SPLINE
SPL {X  -117.449, Y  +780.140, Z    +0.000, E1  +415.491, E3 -83319.411}
SPL {X  -137.837, Y  +752.727, Z    +0.000, E1  +411.385, E3 -83338.899}
SPL {X  -150.415, Y  +726.018, Z    +0.000, E1  +402.769, E3 -83347.774}
SPL {X  -156.153, Y  +706.328, Z    +0.000, E1  +392.414, E3 -83351.466}
SPL {X  -159.178, Y  +687.603, Z    +0.000, E1  +378.267, E3 -83353.444}
SPL {X  -159.915, Y  +676.399, Z    +0.000, E1  +367.484, E3 -83354.014}
SPL {X  -159.990, Y  +669.381, Z    +0.000, E1  +359.965, E3 -83354.114}
SPL {X  -159.990, Y  +666.412, Z    +0.000, E1  +352.765, E3 -83354.146}
SPL {X  -159.990, Y  +662.995, Z    +0.000, E1  +343.976, E3 -83354.248}
SPL {X  -159.990, Y  +658.179, Z    +0.000, E1  +331.312, E3 -83354.485}
SPL {X  -159.990, Y  +652.822, Z    +0.000, E1  +319.345, E3 -83354.899}
SPL {X  -159.990, Y  +646.185, Z    +0.000, E1  +308.728, E3 -83355.638}
SPL {X  -159.990, Y  +632.371, Z    +0.000, E1  +297.040, E3 -83357.991}
SPL {X  -159.990, Y  +579.000, Z    +0.000, E1  +286.931, E3 -83372.863}
SPL {X  -157.725, Y  +355.675, Z    +0.000, E1  +284.959, E3 -83469.821}
SPL {X  -142.593, Y  +309.947, Z    +0.000, E1  +282.426, E3 -83463.485}
SPL {X  -142.198, Y  +309.176, Z    +0.000, E1  +283.218, E3 -83472.293}
ENDSPLINE

SPLINE
SPL {X  -142.352, Y  +309.474, Z    +0.000, E1  +284.206, E3 -83481.987}
ENDSPLINE

SPLINE
SPL {X  -141.553, Y  +307.937, Z    +0.000, E1  +285.290, E3 -83493.003}
SPL {X  -140.562, Y  +306.086, Z    +0.000, E1  +286.440, E3 -83503.697}
SPL {X  -138.743, Y  +302.832, Z    +0.000, E1  +287.062, E3 -83510.494}
SPL {X  -135.531, Y  +297.482, Z    +0.000, E1  +287.444, E3 -83516.329}
SPL {X  -132.271, Y  +292.493, Z    +0.000, E1  +287.844, E3 -83521.847}
SPL {X  -128.837, Y  +287.643, Z    +0.000, E1  +288.283, E3 -83527.285}
SPL {X  -125.941, Y  +283.830, Z    +0.000, E1  +288.683, E3 -83531.584}
SPL {X  -122.669, Y  +279.791, Z    +0.000, E1  +289.119, E3 -83536.078}
SPL {X  -119.730, Y  +276.380, Z    +0.000, E1  +289.584, E3 -83539.866}
SPL {X   -74.058, Y  +240.683, Z    +0.000, E1  +305.011, E3 -83695.582}
ENDSPLINE

SPLINE
SPL {X  -130.401, Y  +289.805, Z    +0.000, E1  +307.505, E3 -83852.553}
SPL {X  -152.244, Y  +333.323, Z    +0.000, E1  +320.871, E3 -83869.365}
SPL {X  -158.218, Y  +358.753, Z    +0.000, E1  +336.397, E3 -83873.537}
SPL {X  -159.681, Y  +372.564, Z    +0.000, E1  +347.981, E3 -83874.589}
SPL {X  -159.987, Y  +381.561, Z    +0.000, E1  +356.806, E3 -83874.885}
SPL {X  -159.990, Y  +384.668, Z    +0.000, E1  +360.183, E3 -83874.911}
SPL {X  -159.990, Y  +387.837, Z    +0.000, E1  +367.342, E3 -83874.951}
SPL {X  -159.990, Y  +393.084, Z    +0.000, E1  +380.137, E3 -83875.161}
SPL {X  -159.990, Y  +401.914, Z    +0.000, E1  +400.147, E3 -83875.855}
SPL {X  -159.990, Y  +414.609, Z    +0.000, E1  +416.791, E3 -83877.592}
SPL {X  -159.990, Y  +464.476, Z    +0.000, E1  +431.765, E3 -83890.393}
SPL {X  -157.643, Y  +698.802, Z    +0.000, E1  +434.751, E3 -83993.407}
SPL {X  -154.470, Y  +713.164, Z    +0.000, E1  +434.425, E3 -84004.996}
SPL {X  -151.032, Y  +724.285, Z    +0.000, E1  +434.102, E3 -84014.800}
SPL {X  -147.134, Y  +734.337, Z    +0.000, E1  +433.686, E3 -84024.437}
SPL {X  -143.804, Y  +741.622, Z    +0.000, E1  +433.324, E3 -84031.825}
SPL {X  -140.603, Y  +747.839, Z    +0.000, E1  +432.964, E3 -84038.341}
SPL {X  -137.184, Y  +753.824, Z    +0.000, E1  +432.574, E3 -84044.778}
SPL {X  -133.762, Y  +759.276, Z    +0.000, E1  +432.150, E3 -84050.831}
SPL {X  -130.927, Y  +763.451, Z    +0.000, E1  +431.785, E3 -84055.526}
SPL {X  -126.852, Y  +768.996, Z    +0.000, E1  +431.276, E3 -84061.757}
SPL {X  -122.512, Y  +774.396, Z    +0.000, E1  +430.640, E3 -84067.866}
SPL {X  -119.782, Y  +777.562, Z    +0.000, E1  +430.221, E3 -84071.373}
SPL {X   -71.924, Y  +814.412, Z    +0.000, E1  +415.124, E3 -84228.243}
ENDSPLINE

SPLINE
SPL {X  -132.255, Y  +761.530, Z    +0.000, E1  +413.203, E3 -84391.413}
SPL {X  -150.415, Y  +726.018, Z    +0.000, E1  +402.769, E3 -84404.917}
SPL {X  -156.153, Y  +706.328, Z    +0.000, E1  +392.414, E3 -84408.609}
SPL {X  -159.178, Y  +687.603, Z    +0.000, E1  +378.267, E3 -84410.587}
SPL {X  -159.974, Y  +673.783, Z    +0.000, E1  +364.843, E3 -84411.209}
SPL {X  -159.990, Y  +669.500, Z    +0.000, E1  +360.000, E3 -84411.256}
SPL {X  -159.990, Y  +667.470, Z    +0.000, E1  +355.588, E3 -84411.274}
SPL {X  -159.990, Y  +662.995, Z    +0.000, E1  +343.976, E3 -84411.391}
SPL {X  -159.990, Y  +658.179, Z    +0.000, E1  +331.312, E3 -84411.628}
SPL {X  -159.990, Y  +652.822, Z    +0.000, E1  +319.345, E3 -84412.042}
SPL {X  -159.990, Y  +646.185, Z    +0.000, E1  +308.728, E3 -84412.781}
SPL {X  -159.990, Y  +632.371, Z    +0.000, E1  +297.040, E3 -84415.134}
SPL {X  -159.990, Y  +579.000, Z    +0.000, E1  +286.931, E3 -84430.006}
SPL {X  -157.725, Y  +355.675, Z    +0.000, E1  +284.959, E3 -84526.964}
SPL {X  -142.593, Y  +309.947, Z    +0.000, E1  +282.426, E3 -84520.628}
SPL {X  -142.198, Y  +309.176, Z    +0.000, E1  +283.218, E3 -84529.436}
ENDSPLINE

SPLINE
SPL {X  -142.352, Y  +309.474, Z    +0.000, E1  +284.206, E3 -84539.130}
ENDSPLINE

SPLINE
SPL {X  -141.553, Y  +307.937, Z    +0.000, E1  +285.290, E3 -84550.146}
SPL {X  -140.562, Y  +306.086, Z    +0.000, E1  +286.440, E3 -84560.839}
SPL {X  -138.743, Y  +302.832, Z    +0.000, E1  +287.062, E3 -84567.637}
SPL {X  -135.531, Y  +297.482, Z    +0.000, E1  +287.444, E3 -84573.471}
SPL {X  -132.271, Y  +292.493, Z    +0.000, E1  +287.844, E3 -84578.990}
SPL {X  -128.837, Y  +287.643, Z    +0.000, E1  +288.283, E3 -84584.428}
SPL {X  -124.965, Y  +282.598, Z    +0.000, E1  +288.800, E3 -84590.089}
SPL {X  -120.791, Y  +277.589, Z    +0.000, E1  +289.397, E3 -84595.662}
SPL {X   -74.058, Y  +240.683, Z    +0.000, E1  +305.011, E3 -84752.725}
ENDSPLINE

SPLINE
SPL {X  -130.401, Y  +289.805, Z    +0.000, E1  +307.505, E3 -84909.696}
SPL {X  -148.502, Y  +322.968, Z    +0.000, E1  +316.497, E3 -84924.016}
SPL {X  -154.800, Y  +342.080, Z    +0.000, E1  +325.471, E3 -84928.320}
SPL {X  -158.218, Y  +358.753, Z    +0.000, E1  +336.397, E3 -84930.680}
SPL {X  -159.681, Y  +372.564, Z    +0.000, E1  +347.981, E3 -84931.731}
SPL {X  -159.987, Y  +381.561, Z    +0.000, E1  +356.806, E3 -84932.028}
SPL {X  -159.990, Y  +384.668, Z    +0.000, E1  +360.183, E3 -84932.054}
SPL {X  -159.990, Y  +387.837, Z    +0.000, E1  +367.342, E3 -84932.094}
SPL {X  -159.990, Y  +393.084, Z    +0.000, E1  +380.137, E3 -84932.304}
SPL {X  -159.990, Y  +401.914, Z    +0.000, E1  +400.147, E3 -84932.998}
SPL {X  -159.990, Y  +414.609, Z    +0.000, E1  +416.791, E3 -84934.735}
SPL {X  -159.990, Y  +464.476, Z    +0.000, E1  +431.765, E3 -84947.536}
SPL {X  -157.643, Y  +698.802, Z    +0.000, E1  +434.751, E3 -85050.550}
SPL {X  -154.470, Y  +713.164, Z    +0.000, E1  +434.425, E3 -85062.139}
SPL {X  -151.032, Y  +724.285, Z    +0.000, E1  +434.102, E3 -85071.943}
SPL {X  -147.134, Y  +734.337, Z    +0.000, E1  +433.686, E3 -85081.580}
SPL {X  -143.804, Y  +741.622, Z    +0.000, E1  +433.324, E3 -85088.968}
SPL {X  -140.603, Y  +747.839, Z    +0.000, E1  +432.964, E3 -85095.484}
SPL {X  -137.184, Y  +753.824, Z    +0.000, E1  +432.574, E3 -85101.920}
SPL {X  -133.762, Y  +759.276, Z    +0.000, E1  +432.150, E3 -85107.974}
SPL {X  -130.927, Y  +763.451, Z    +0.000, E1  +431.785, E3 -85112.669}
SPL {X  -126.852, Y  +768.996, Z    +0.000, E1  +431.276, E3 -85118.900}
SPL {X  -122.512, Y  +774.396, Z    +0.000, E1  +430.640, E3 -85125.009}
SPL {X  -119.782, Y  +777.562, Z    +0.000, E1  +430.221, E3 -85128.516}
SPL {X   -71.924, Y  +814.412, Z    +0.000, E1  +415.124, E3 -85285.386}
ENDSPLINE

SPLINE
SPL {X  -132.255, Y  +761.530, Z    +0.000, E1  +413.203, E3 -85448.556}
SPL {X  -150.415, Y  +726.018, Z    +0.000, E1  +402.769, E3 -85462.060}
SPL {X  -156.153, Y  +706.328, Z    +0.000, E1  +392.414, E3 -85465.752}
SPL {X  -159.178, Y  +687.603, Z    +0.000, E1  +378.267, E3 -85467.730}
SPL {X  -159.915, Y  +676.399, Z    +0.000, E1  +367.484, E3 -85468.300}
SPL {X  -159.990, Y  +669.585, Z    +0.000, E1  +360.185, E3 -85468.399}
SPL {X  -159.990, Y  +667.470, Z    +0.000, E1  +355.588, E3 -85468.417}
SPL {X  -159.990, Y  +662.995, Z    +0.000, E1  +343.976, E3 -85468.534}
SPL {X  -159.990, Y  +658.179, Z    +0.000, E1  +331.312, E3 -85468.770}
SPL {X  -159.990, Y  +652.822, Z    +0.000, E1  +319.345, E3 -85469.185}
SPL {X  -159.990, Y  +646.185, Z    +0.000, E1  +308.728, E3 -85469.924}
SPL {X  -159.990, Y  +632.371, Z    +0.000, E1  +297.040, E3 -85472.276}
SPL {X  -159.990, Y  +579.000, Z    +0.000, E1  +286.931, E3 -85487.149}
SPL {X  -157.725, Y  +355.675, Z    +0.000, E1  +284.959, E3 -85584.107}
SPL {X  -142.593, Y  +309.947, Z    +0.000, E1  +282.426, E3 -85577.770}
SPL {X  -142.198, Y  +309.176, Z    +0.000, E1  +283.218, E3 -85586.579}
ENDSPLINE

SPLINE
SPL {X  -142.352, Y  +309.474, Z    +0.000, E1  +284.206, E3 -85596.273}
ENDSPLINE

SPLINE
SPL {X  -141.553, Y  +307.937, Z    +0.000, E1  +285.290, E3 -85607.288}
SPL {X  -140.562, Y  +306.086, Z    +0.000, E1  +286.440, E3 -85617.982}
SPL {X  -138.743, Y  +302.832, Z    +0.000, E1  +287.062, E3 -85624.780}
SPL {X  -135.531, Y  +297.482, Z    +0.000, E1  +287.444, E3 -85630.614}
SPL {X  -132.271, Y  +292.493, Z    +0.000, E1  +287.844, E3 -85636.133}
SPL {X  -128.837, Y  +287.643, Z    +0.000, E1  +288.283, E3 -85641.570}
SPL {X  -124.965, Y  +282.598, Z    +0.000, E1  +288.800, E3 -85647.232}
SPL {X  -120.791, Y  +277.589, Z    +0.000, E1  +289.397, E3 -85652.805}
SPL {X   -74.058, Y  +240.683, Z    +0.000, E1  +305.011, E3 -85809.868}
ENDSPLINE

SPLINE
SPL {X  -130.401, Y  +289.805, Z    +0.000, E1  +307.505, E3 -85966.839}
SPL {X  -148.502, Y  +322.968, Z    +0.000, E1  +316.497, E3 -85981.159}
SPL {X  -154.800, Y  +342.080, Z    +0.000, E1  +325.471, E3 -85985.463}
SPL {X  -158.218, Y  +358.753, Z    +0.000, E1  +336.397, E3 -85987.823}
SPL {X  -159.681, Y  +372.564, Z    +0.000, E1  +347.981, E3 -85988.874}
SPL {X  -159.987, Y  +381.561, Z    +0.000, E1  +356.806, E3 -85989.171}
SPL {X  -159.990, Y  +384.668, Z    +0.000, E1  +360.183, E3 -85989.196}
SPL {X  -159.990, Y  +387.837, Z    +0.000, E1  +367.342, E3 -85989.237}
SPL {X  -159.990, Y  +393.084, Z    +0.000, E1  +380.137, E3 -85989.447}
SPL {X  -159.990, Y  +401.914, Z    +0.000, E1  +400.147, E3 -85990.141}
SPL {X  -159.990, Y  +414.609, Z    +0.000, E1  +416.791, E3 -85991.877}
SPL {X  -159.990, Y  +464.476, Z    +0.000, E1  +431.765, E3 -86004.678}
SPL {X  -157.643, Y  +698.802, Z    +0.000, E1  +434.751, E3 -86107.693}
SPL {X  -154.470, Y  +713.164, Z    +0.000, E1  +434.425, E3 -86119.282}
SPL {X  -151.032, Y  +724.285, Z    +0.000, E1  +434.102, E3 -86129.086}
SPL {X  -147.134, Y  +734.337, Z    +0.000, E1  +433.686, E3 -86138.723}
SPL {X  -143.804, Y  +741.622, Z    +0.000, E1  +433.324, E3 -86146.111}
SPL {X  -140.603, Y  +747.839, Z    +0.000, E1  +432.964, E3 -86152.627}
SPL {X  -137.184, Y  +753.824, Z    +0.000, E1  +432.574, E3 -86159.063}
SPL {X  -133.762, Y  +759.276, Z    +0.000, E1  +432.150, E3 -86165.117}
SPL {X  -130.927, Y  +763.451, Z    +0.000, E1  +431.785, E3 -86169.812}
SPL {X  -128.105, Y  +767.343, Z    +0.000, E1  +431.419, E3 -86174.200}
SPL {X  -124.554, Y  +771.914, Z    +0.000, E1  +430.935, E3 -86179.371}
SPL {X  -120.687, Y  +776.531, Z    +0.000, E1  +430.379, E3 -86184.505}
SPL {X   -71.924, Y  +814.412, Z    +0.000, E1  +415.124, E3 -86342.529}
ENDSPLINE

SPLINE
SPL {X  -132.255, Y  +761.530, Z    +0.000, E1  +413.203, E3 -86505.699}
SPL {X  -150.415, Y  +726.018, Z    +0.000, E1  +402.769, E3 -86519.203}
SPL {X  -156.153, Y  +706.328, Z    +0.000, E1  +392.414, E3 -86522.895}
SPL {X  -159.178, Y  +687.603, Z    +0.000, E1  +378.267, E3 -86524.873}
SPL {X  -159.974, Y  +673.783, Z    +0.000, E1  +364.843, E3 -86525.495}
SPL {X  -159.990, Y  +669.500, Z    +0.000, E1  +360.000, E3 -86525.542}
SPL {X  -159.990, Y  +667.470, Z    +0.000, E1  +355.588, E3 -86525.560}
SPL {X  -159.990, Y  +662.995, Z    +0.000, E1  +343.976, E3 -86525.677}
SPL {X  -159.990, Y  +658.179, Z    +0.000, E1  +331.312, E3 -86525.913}
SPL {X  -159.990, Y  +652.822, Z    +0.000, E1  +319.345, E3 -86526.328}
SPL {X  -159.990, Y  +646.185, Z    +0.000, E1  +308.728, E3 -86527.067}
SPL {X  -159.990, Y  +636.375, Z    +0.000, E1  +299.286, E3 -86528.506}
SPL {X  -159.990, Y  +617.374, Z    +0.000, E1  +291.478, E3 -86532.833}
SPL {X  -159.990, Y  +579.000, Z    +0.000, E1  +286.931, E3 -86544.292}
SPL {X  -157.725, Y  +355.675, Z    +0.000, E1  +284.959, E3 -86641.250}
SPL {X  -142.593, Y  +309.947, Z    +0.000, E1  +282.426, E3 -86634.913}
SPL {X  -142.198, Y  +309.176, Z    +0.000, E1  +283.218, E3 -86643.722}
ENDSPLINE

SPLINE
SPL {X  -142.352, Y  +309.474, Z    +0.000, E1  +284.206, E3 -86653.415}
ENDSPLINE

SPLINE
SPL {X  -141.929, Y  +308.657, Z    +0.000, E1  +285.131, E3 -86662.501}
SPL {X  -140.635, Y  +306.221, Z    +0.000, E1  +286.163, E3 -86672.913}
SPL {X  -138.743, Y  +302.832, Z    +0.000, E1  +287.062, E3 -86681.923}
SPL {X  -135.531, Y  +297.482, Z    +0.000, E1  +287.444, E3 -86687.757}
SPL {X  -132.271, Y  +292.493, Z    +0.000, E1  +287.844, E3 -86693.276}
SPL {X  -128.837, Y  +287.643, Z    +0.000, E1  +288.283, E3 -86698.713}
SPL {X  -125.941, Y  +283.830, Z    +0.000, E1  +288.683, E3 -86703.013}
SPL {X  -124.080, Y  +281.501, Z    +0.000, E1  +288.943, E3 -86705.624}
SPL {X  -120.791, Y  +277.589, Z    +0.000, E1  +289.397, E3 -86709.948}
SPL {X   -74.058, Y  +240.683, Z    +0.000, E1  +305.011, E3 -86867.011}
ENDSPLINE

SPLINE
SPL {X  -130.401, Y  +289.805, Z    +0.000, E1  +307.505, E3 -87023.982}
SPL {X  -152.244, Y  +333.323, Z    +0.000, E1  +320.871, E3 -87040.793}
SPL {X  -158.218, Y  +358.753, Z    +0.000, E1  +336.397, E3 -87044.966}
SPL {X  -159.681, Y  +372.564, Z    +0.000, E1  +347.981, E3 -87046.017}
SPL {X  -159.987, Y  +381.561, Z    +0.000, E1  +356.806, E3 -87046.314}
SPL {X  -159.990, Y  +384.668, Z    +0.000, E1  +360.183, E3 -87046.339}
SPL {X  -159.990, Y  +387.837, Z    +0.000, E1  +367.342, E3 -87046.380}
SPL {X  -159.990, Y  +393.084, Z    +0.000, E1  +380.137, E3 -87046.590}
SPL {X  -159.990, Y  +401.914, Z    +0.000, E1  +400.147, E3 -87047.283}
SPL {X  -159.990, Y  +414.609, Z    +0.000, E1  +416.791, E3 -87049.020}
SPL {X  -159.990, Y  +464.476, Z    +0.000, E1  +431.765, E3 -87061.821}
SPL {X  -158.553, Y  +692.895, Z    +0.000, E1  +434.809, E3 -87160.585}
SPL {X  -156.740, Y  +703.585, Z    +0.000, E1  +434.640, E3 -87168.589}
SPL {X  -154.470, Y  +713.164, Z    +0.000, E1  +434.425, E3 -87176.425}
SPL {X  -151.032, Y  +724.285, Z    +0.000, E1  +434.102, E3 -87186.228}
SPL {X  -147.134, Y  +734.337, Z    +0.000, E1  +433.686, E3 -87195.866}
SPL {X  -143.804, Y  +741.622, Z    +0.000, E1  +433.324, E3 -87203.254}
SPL {X  -140.603, Y  +747.839, Z    +0.000, E1  +432.964, E3 -87209.769}
SPL {X  -137.184, Y  +753.824, Z    +0.000, E1  +432.574, E3 -87216.206}
SPL {X  -133.762, Y  +759.276, Z    +0.000, E1  +432.150, E3 -87222.260}
SPL {X  -130.927, Y  +763.451, Z    +0.000, E1  +431.785, E3 -87226.954}
SPL {X  -126.852, Y  +768.996, Z    +0.000, E1  +431.276, E3 -87233.185}
SPL {X  -122.512, Y  +774.396, Z    +0.000, E1  +430.640, E3 -87239.295}
SPL {X  -119.782, Y  +777.562, Z    +0.000, E1  +430.221, E3 -87242.802}
SPL {X   -71.924, Y  +814.412, Z    +0.000, E1  +415.124, E3 -87399.672}
ENDSPLINE

SPLINE
SPL {X  -132.255, Y  +761.530, Z    +0.000, E1  +413.203, E3 -87562.842}
SPL {X  -150.415, Y  +726.018, Z    +0.000, E1  +402.769, E3 -87576.346}
SPL {X  -156.153, Y  +706.328, Z    +0.000, E1  +392.414, E3 -87580.038}
SPL {X  -159.178, Y  +687.603, Z    +0.000, E1  +378.267, E3 -87582.016}
SPL {X  -159.974, Y  +673.783, Z    +0.000, E1  +364.843, E3 -87582.637}
SPL {X  -159.990, Y  +669.500, Z    +0.000, E1  +360.000, E3 -87582.685}
SPL {X  -159.990, Y  +667.470, Z    +0.000, E1  +355.588, E3 -87582.703}
SPL {X  -159.990, Y  +662.995, Z    +0.000, E1  +343.976, E3 -87582.819}
SPL {X  -159.990, Y  +658.179, Z    +0.000, E1  +331.312, E3 -87583.056}
SPL {X  -159.990, Y  +652.822, Z    +0.000, E1  +319.345, E3 -87583.471}
SPL {X  -159.990, Y  +646.185, Z    +0.000, E1  +308.728, E3 -87584.210}
SPL {X  -159.990, Y  +636.375, Z    +0.000, E1  +299.286, E3 -87585.649}
SPL {X  -159.990, Y  +617.374, Z    +0.000, E1  +291.478, E3 -87589.975}
SPL {X  -159.990, Y  +579.000, Z    +0.000, E1  +286.931, E3 -87601.434}
SPL {X  -157.725, Y  +355.675, Z    +0.000, E1  +284.959, E3 -87698.393}
SPL {X  -142.593, Y  +309.947, Z    +0.000, E1  +282.426, E3 -87692.056}
SPL {X  -142.198, Y  +309.176, Z    +0.000, E1  +283.218, E3 -87700.865}
ENDSPLINE

SPLINE
SPL {X  -142.352, Y  +309.474, Z    +0.000, E1  +284.206, E3 -87710.558}
ENDSPLINE

SPLINE
SPL {X  -141.553, Y  +307.937, Z    +0.000, E1  +285.290, E3 -87721.574}
SPL {X  -140.562, Y  +306.086, Z    +0.000, E1  +286.440, E3 -87732.268}
SPL {X  -138.743, Y  +302.832, Z    +0.000, E1  +287.062, E3 -87739.065}
SPL {X  -135.531, Y  +297.482, Z    +0.000, E1  +287.444, E3 -87744.900}
SPL {X  -132.271, Y  +292.493, Z    +0.000, E1  +287.844, E3 -87750.418}
SPL {X  -128.837, Y  +287.643, Z    +0.000, E1  +288.283, E3 -87755.856}
SPL {X  -125.941, Y  +283.830, Z    +0.000, E1  +288.683, E3 -87760.156}
SPL {X  -124.080, Y  +281.501, Z    +0.000, E1  +288.943, E3 -87762.766}
SPL {X  -120.791, Y  +277.589, Z    +0.000, E1  +289.397, E3 -87767.091}
SPL {X   -74.058, Y  +240.683, Z    +0.000, E1  +305.011, E3 -87924.154}
ENDSPLINE

SPLINE
SPL {X  -130.401, Y  +289.805, Z    +0.000, E1  +307.505, E3 -88081.125}
SPL {X  -148.502, Y  +322.968, Z    +0.000, E1  +316.497, E3 -88095.445}
SPL {X  -154.800, Y  +342.080, Z    +0.000, E1  +325.471, E3 -88099.749}
SPL {X  -158.218, Y  +358.753, Z    +0.000, E1  +336.397, E3 -88102.108}
SPL {X  -159.681, Y  +372.564, Z    +0.000, E1  +347.981, E3 -88103.160}
SPL {X  -159.987, Y  +381.561, Z    +0.000, E1  +356.806, E3 -88103.456}
SPL {X  -159.990, Y  +384.668, Z    +0.000, E1  +360.183, E3 -88103.482}
SPL {X  -159.990, Y  +387.837, Z    +0.000, E1  +367.342, E3 -88103.523}
SPL {X  -159.990, Y  +393.084, Z    +0.000, E1  +380.137, E3 -88103.733}
SPL {X  -159.990, Y  +401.914, Z    +0.000, E1  +400.147, E3 -88104.426}
SPL {X  -159.990, Y  +414.609, Z    +0.000, E1  +416.791, E3 -88106.163}
SPL {X  -159.990, Y  +464.476, Z    +0.000, E1  +431.765, E3 -88118.964}
SPL {X  -157.643, Y  +698.802, Z    +0.000, E1  +434.751, E3 -88221.979}
SPL {X  -154.470, Y  +713.164, Z    +0.000, E1  +434.425, E3 -88233.568}
SPL {X  -152.098, Y  +721.129, Z    +0.000, E1  +434.190, E3 -88240.540}
SPL {X  -148.128, Y  +731.956, Z    +0.000, E1  +433.814, E3 -88250.621}
SPL {X  -143.804, Y  +741.622, Z    +0.000, E1  +433.324, E3 -88260.397}
SPL {X  -140.603, Y  +747.839, Z    +0.000, E1  +432.964, E3 -88266.912}
SPL {X  -137.184, Y  +753.824, Z    +0.000, E1  +432.574, E3 -88273.349}
SPL {X  -133.762, Y  +759.276, Z    +0.000, E1  +432.150, E3 -88279.403}
SPL {X  -130.927, Y  +763.451, Z    +0.000, E1  +431.785, E3 -88284.097}
SPL {X  -128.105, Y  +767.343, Z    +0.000, E1  +431.419, E3 -88288.486}
SPL {X  -124.554, Y  +771.914, Z    +0.000, E1  +430.935, E3 -88293.657}
SPL {X  -120.687, Y  +776.531, Z    +0.000, E1  +430.379, E3 -88298.790}
SPL {X   -71.924, Y  +814.412, Z    +0.000, E1  +415.124, E3 -88456.815}
ENDSPLINE

SPLINE
SPL {X  -132.255, Y  +761.530, Z    +0.000, E1  +413.203, E3 -88619.984}
SPL {X  -150.415, Y  +726.018, Z    +0.000, E1  +402.769, E3 -88633.488}
SPL {X  -157.206, Y  +701.216, Z    +0.000, E1  +389.056, E3 -88637.827}
SPL {X  -159.772, Y  +679.843, Z    +0.000, E1  +371.089, E3 -88639.591}
SPL {X  -159.990, Y  +669.381, Z    +0.000, E1  +359.965, E3 -88639.828}
SPL {X  -159.990, Y  +666.412, Z    +0.000, E1  +352.765, E3 -88639.860}
SPL {X  -159.990, Y  +662.995, Z    +0.000, E1  +343.976, E3 -88639.962}
SPL {X  -159.990, Y  +658.179, Z    +0.000, E1  +331.312, E3 -88640.199}
SPL {X  -159.990, Y  +652.822, Z    +0.000, E1  +319.345, E3 -88640.614}
SPL {X  -159.990, Y  +646.185, Z    +0.000, E1  +308.728, E3 -88641.352}
SPL {X  -159.990, Y  +632.371, Z    +0.000, E1  +297.040, E3 -88643.705}
SPL {X  -159.990, Y  +579.000, Z    +0.000, E1  +286.931, E3 -88658.577}
SPL {X  -157.725, Y  +355.675, Z    +0.000, E1  +284.959, E3 -88755.536}
SPL {X  -142.593, Y  +309.947, Z    +0.000, E1  +282.426, E3 -88749.199}
SPL {X  -142.198, Y  +309.176, Z    +0.000, E1  +283.218, E3 -88758.008}
ENDSPLINE

SPLINE
SPL {X  -142.352, Y  +309.474, Z    +0.000, E1  +284.206, E3 -88767.701}
ENDSPLINE

SPLINE
SPL {X  -141.929, Y  +308.657, Z    +0.000, E1  +285.131, E3 -88776.786}
SPL {X  -140.635, Y  +306.221, Z    +0.000, E1  +286.163, E3 -88787.199}
SPL {X  -138.743, Y  +302.832, Z    +0.000, E1  +287.062, E3 -88796.208}
SPL {X  -135.531, Y  +297.482, Z    +0.000, E1  +287.444, E3 -88802.043}
SPL {X  -132.271, Y  +292.493, Z    +0.000, E1  +287.844, E3 -88807.561}
SPL {X  -128.837, Y  +287.643, Z    +0.000, E1  +288.283, E3 -88812.999}
SPL {X  -124.965, Y  +282.598, Z    +0.000, E1  +288.800, E3 -88818.661}
SPL {X  -120.791, Y  +277.589, Z    +0.000, E1  +289.397, E3 -88824.234}
SPL {X   -74.058, Y  +240.683, Z    +0.000, E1  +305.011, E3 -88981.297}
ENDSPLINE

SPLINE
SPL {X  -130.401, Y  +289.805, Z    +0.000, E1  +307.505, E3 -89138.267}
SPL {X  -148.502, Y  +322.968, Z    +0.000, E1  +316.497, E3 -89152.588}
SPL {X  -154.800, Y  +342.080, Z    +0.000, E1  +325.471, E3 -89156.891}
SPL {X  -158.218, Y  +358.753, Z    +0.000, E1  +336.397, E3 -89159.251}
SPL {X  -159.681, Y  +372.564, Z    +0.000, E1  +347.981, E3 -89160.303}
SPL {X  -159.987, Y  +381.561, Z    +0.000, E1  +356.806, E3 -89160.599}
SPL {X  -159.990, Y  +384.668, Z    +0.000, E1  +360.183, E3 -89160.625}
SPL {X  -159.990, Y  +387.837, Z    +0.000, E1  +367.342, E3 -89160.666}
SPL {X  -159.990, Y  +393.084, Z    +0.000, E1  +380.137, E3 -89160.876}
SPL {X  -159.990, Y  +401.914, Z    +0.000, E1  +400.147, E3 -89161.569}
SPL {X  -159.990, Y  +414.609, Z    +0.000, E1  +416.791, E3 -89163.306}
SPL {X  -159.990, Y  +464.476, Z    +0.000, E1  +431.765, E3 -89176.107}
SPL {X  -157.643, Y  +698.802, Z    +0.000, E1  +434.751, E3 -89279.122}
SPL {X  -154.470, Y  +713.164, Z    +0.000, E1  +434.425, E3 -89290.710}
SPL {X  -151.032, Y  +724.285, Z    +0.000, E1  +434.102, E3 -89300.514}
SPL {X  -147.134, Y  +734.337, Z    +0.000, E1  +433.686, E3 -89310.152}
SPL {X  -143.804, Y  +741.622, Z    +0.000, E1  +433.324, E3 -89317.540}
SPL {X  -140.603, Y  +747.839, Z    +0.000, E1  +432.964, E3 -89324.055}
SPL {X  -137.184, Y  +753.824, Z    +0.000, E1  +432.574, E3 -89330.492}
SPL {X  -133.762, Y  +759.276, Z    +0.000, E1  +432.150, E3 -89336.546}
SPL {X  -130.927, Y  +763.451, Z    +0.000, E1  +431.785, E3 -89341.240}
SPL {X  -128.105, Y  +767.343, Z    +0.000, E1  +431.419, E3 -89345.629}
SPL {X  -124.554, Y  +771.914, Z    +0.000, E1  +430.935, E3 -89350.800}
SPL {X  -120.892, Y  +776.295, Z    +0.000, E1  +430.404, E3 -89355.684}
SPL {X  -118.039, Y  +779.498, Z    +0.000, E1  +429.949, E3 -89359.202}
SPL {X   -71.924, Y  +814.412, Z    +0.000, E1  +415.124, E3 -89513.958}
ENDSPLINE

SPLINE
SPL {X  -132.255, Y  +761.530, Z    +0.000, E1  +413.203, E3 -89677.127}
SPL {X  -150.415, Y  +726.018, Z    +0.000, E1  +402.769, E3 -89690.631}
SPL {X  -156.153, Y  +706.328, Z    +0.000, E1  +392.414, E3 -89694.323}
SPL {X  -159.178, Y  +687.603, Z    +0.000, E1  +378.267, E3 -89696.301}
SPL {X  -159.974, Y  +673.783, Z    +0.000, E1  +364.843, E3 -89696.923}
SPL {X  -159.990, Y  +669.500, Z    +0.000, E1  +360.000, E3 -89696.971}
SPL {X  -159.990, Y  +667.470, Z    +0.000, E1  +355.588, E3 -89696.989}
SPL {X  -159.990, Y  +662.995, Z    +0.000, E1  +343.976, E3 -89697.105}
SPL {X  -159.990, Y  +658.179, Z    +0.000, E1  +331.312, E3 -89697.342}
SPL {X  -159.990, Y  +652.822, Z    +0.000, E1  +319.345, E3 -89697.757}
SPL {X  -159.990, Y  +646.185, Z    +0.000, E1  +308.728, E3 -89698.495}
SPL {X  -159.990, Y  +636.375, Z    +0.000, E1  +299.286, E3 -89699.935}
SPL {X  -159.990, Y  +617.374, Z    +0.000, E1  +291.478, E3 -89704.261}
SPL {X  -159.990, Y  +579.000, Z    +0.000, E1  +286.931, E3 -89715.720}
SPL {X  -157.725, Y  +355.675, Z    +0.000, E1  +284.959, E3 -89812.678}
SPL {X  -142.593, Y  +309.947, Z    +0.000, E1  +282.426, E3 -89806.342}
SPL {X  -142.198, Y  +309.176, Z    +0.000, E1  +283.218, E3 -89815.150}
ENDSPLINE

SPLINE
SPL {X  -142.352, Y  +309.474, Z    +0.000, E1  +284.206, E3 -89824.844}
ENDSPLINE

SPLINE
SPL {X  -141.553, Y  +307.937, Z    +0.000, E1  +285.290, E3 -89835.860}
SPL {X  -140.562, Y  +306.086, Z    +0.000, E1  +286.440, E3 -89846.554}
SPL {X  -138.743, Y  +302.832, Z    +0.000, E1  +287.062, E3 -89853.351}
SPL {X  -135.531, Y  +297.482, Z    +0.000, E1  +287.444, E3 -89859.186}
SPL {X  -132.271, Y  +292.493, Z    +0.000, E1  +287.844, E3 -89864.704}
SPL {X  -128.837, Y  +287.643, Z    +0.000, E1  +288.283, E3 -89870.142}
SPL {X  -125.941, Y  +283.830, Z    +0.000, E1  +288.683, E3 -89874.442}
SPL {X  -124.080, Y  +281.501, Z    +0.000, E1  +288.943, E3 -89877.052}
SPL {X  -120.791, Y  +277.589, Z    +0.000, E1  +289.397, E3 -89881.376}
SPL {X   -74.058, Y  +240.683, Z    +0.000, E1  +305.011, E3 -90038.439}
ENDSPLINE

SPLINE
SPL {X  -130.401, Y  +289.805, Z    +0.000, E1  +307.505, E3 -90195.410}
SPL {X  -152.244, Y  +333.323, Z    +0.000, E1  +320.871, E3 -90212.222}
SPL {X  -158.218, Y  +358.753, Z    +0.000, E1  +336.397, E3 -90216.394}
SPL {X  -159.681, Y  +372.564, Z    +0.000, E1  +347.981, E3 -90217.446}
SPL {X  -159.987, Y  +381.561, Z    +0.000, E1  +356.806, E3 -90217.742}
SPL {X  -159.990, Y  +384.668, Z    +0.000, E1  +360.183, E3 -90217.768}
SPL {X  -159.990, Y  +387.837, Z    +0.000, E1  +367.342, E3 -90217.809}
SPL {X  -159.990, Y  +393.084, Z    +0.000, E1  +380.137, E3 -90218.018}
SPL {X  -159.990, Y  +401.914, Z    +0.000, E1  +400.147, E3 -90218.712}
SPL {X  -159.990, Y  +414.609, Z    +0.000, E1  +416.791, E3 -90220.449}
SPL {X  -159.990, Y  +464.476, Z    +0.000, E1  +431.765, E3 -90233.250}
SPL {X  -157.643, Y  +698.802, Z    +0.000, E1  +434.751, E3 -90336.265}
SPL {X  -154.470, Y  +713.164, Z    +0.000, E1  +434.425, E3 -90347.853}
SPL {X  -152.098, Y  +721.129, Z    +0.000, E1  +434.190, E3 -90354.825}
SPL {X  -148.128, Y  +731.956, Z    +0.000, E1  +433.814, E3 -90364.906}
SPL {X  -143.804, Y  +741.622, Z    +0.000, E1  +433.324, E3 -90374.682}
SPL {X  -140.603, Y  +747.839, Z    +0.000, E1  +432.964, E3 -90381.198}
SPL {X  -137.184, Y  +753.824, Z    +0.000, E1  +432.574, E3 -90387.635}
SPL {X  -133.762, Y  +759.276, Z    +0.000, E1  +432.150, E3 -90393.688}
SPL {X  -130.927, Y  +763.451, Z    +0.000, E1  +431.785, E3 -90398.383}
SPL {X  -128.105, Y  +767.343, Z    +0.000, E1  +431.419, E3 -90402.772}
SPL {X  -125.461, Y  +770.778, Z    +0.000, E1  +431.046, E3 -90406.685}
SPL {X  -122.512, Y  +774.396, Z    +0.000, E1  +430.640, E3 -90410.723}
SPL {X  -119.782, Y  +777.562, Z    +0.000, E1  +430.221, E3 -90414.230}
SPL {X   -71.924, Y  +814.412, Z    +0.000, E1  +415.124, E3 -90571.100}
ENDSPLINE

SPLINE
SPL {X  -132.255, Y  +761.530, Z    +0.000, E1  +413.203, E3 -90734.270}
SPL {X  -150.415, Y  +726.018, Z    +0.000, E1  +402.769, E3 -90747.774}
SPL {X  -156.153, Y  +706.328, Z    +0.000, E1  +392.414, E3 -90751.466}
SPL {X  -159.178, Y  +687.603, Z    +0.000, E1  +378.267, E3 -90753.444}
SPL {X  -159.915, Y  +676.399, Z    +0.000, E1  +367.484, E3 -90754.014}
SPL {X  -159.990, Y  +669.585, Z    +0.000, E1  +360.185, E3 -90754.113}
SPL {X  -159.990, Y  +667.470, Z    +0.000, E1  +355.588, E3 -90754.132}
SPL {X  -159.990, Y  +662.995, Z    +0.000, E1  +343.976, E3 -90754.248}
SPL {X  -159.990, Y  +658.179, Z    +0.000, E1  +331.312, E3 -90754.485}
SPL {X  -159.990, Y  +652.822, Z    +0.000, E1  +319.345, E3 -90754.899}
SPL {X  -159.990, Y  +646.185, Z    +0.000, E1  +308.728, E3 -90755.638}
SPL {X  -159.990, Y  +636.375, Z    +0.000, E1  +299.286, E3 -90757.078}
SPL {X  -159.990, Y  +617.374, Z    +0.000, E1  +291.478, E3 -90761.404}
SPL {X  -159.990, Y  +579.000, Z    +0.000, E1  +286.931, E3 -90772.863}
SPL {X  -157.725, Y  +355.675, Z    +0.000, E1  +284.959, E3 -90869.821}
SPL {X  -142.593, Y  +309.947, Z    +0.000, E1  +282.426, E3 -90863.485}
SPL {X  -142.198, Y  +309.176, Z    +0.000, E1  +283.218, E3 -90872.293}
ENDSPLINE

SPLINE
SPL {X  -142.352, Y  +309.474, Z    +0.000, E1  +284.206, E3 -90881.987}
ENDSPLINE

SPLINE
SPL {X  -141.929, Y  +308.657, Z    +0.000, E1  +285.131, E3 -90891.072}
SPL {X  -140.635, Y  +306.221, Z    +0.000, E1  +286.163, E3 -90901.484}
SPL {X  -138.743, Y  +302.832, Z    +0.000, E1  +287.062, E3 -90910.494}
SPL {X  -135.531, Y  +297.482, Z    +0.000, E1  +287.444, E3 -90916.329}
SPL {X  -132.271, Y  +292.493, Z    +0.000, E1  +287.844, E3 -90921.847}
SPL {X  -128.837, Y  +287.643, Z    +0.000, E1  +288.283, E3 -90927.285}
SPL {X  -125.941, Y  +283.830, Z    +0.000, E1  +288.683, E3 -90931.584}
SPL {X  -122.669, Y  +279.791, Z    +0.000, E1  +289.119, E3 -90936.078}
SPL {X  -119.730, Y  +276.380, Z    +0.000, E1  +289.584, E3 -90939.866}
SPL {X   -74.058, Y  +240.683, Z    +0.000, E1  +305.011, E3 -91095.582}
ENDSPLINE

SPLINE
SPL {X  -130.401, Y  +289.805, Z    +0.000, E1  +307.505, E3 -91252.553}
SPL {X  -148.502, Y  +322.968, Z    +0.000, E1  +316.497, E3 -91266.873}
SPL {X  -154.800, Y  +342.080, Z    +0.000, E1  +325.471, E3 -91271.177}
SPL {X  -158.218, Y  +358.753, Z    +0.000, E1  +336.397, E3 -91273.537}
SPL {X  -159.681, Y  +372.564, Z    +0.000, E1  +347.981, E3 -91274.589}
SPL {X  -159.987, Y  +381.561, Z    +0.000, E1  +356.806, E3 -91274.885}
SPL {X  -159.990, Y  +384.668, Z    +0.000, E1  +360.183, E3 -91274.911}
SPL {X  -159.990, Y  +387.837, Z    +0.000, E1  +367.342, E3 -91274.951}
SPL {X  -159.990, Y  +393.084, Z    +0.000, E1  +380.137, E3 -91275.161}
SPL {X  -159.990, Y  +401.914, Z    +0.000, E1  +400.147, E3 -91275.855}
SPL {X  -159.990, Y  +414.609, Z    +0.000, E1  +416.791, E3 -91277.592}
SPL {X  -159.990, Y  +464.476, Z    +0.000, E1  +431.765, E3 -91290.393}
SPL {X  -157.643, Y  +698.802, Z    +0.000, E1  +434.751, E3 -91393.407}
SPL {X  -154.470, Y  +713.164, Z    +0.000, E1  +434.425, E3 -91404.996}
SPL {X  -151.032, Y  +724.285, Z    +0.000, E1  +434.102, E3 -91414.800}
SPL {X  -147.134, Y  +734.337, Z    +0.000, E1  +433.686, E3 -91424.437}
SPL {X  -143.804, Y  +741.622, Z    +0.000, E1  +433.324, E3 -91431.825}
SPL {X  -140.603, Y  +747.839, Z    +0.000, E1  +432.964, E3 -91438.341}
SPL {X  -137.184, Y  +753.824, Z    +0.000, E1  +432.574, E3 -91444.778}
SPL {X  -133.762, Y  +759.276, Z    +0.000, E1  +432.150, E3 -91450.831}
SPL {X  -130.927, Y  +763.451, Z    +0.000, E1  +431.785, E3 -91455.526}
SPL {X  -128.105, Y  +767.343, Z    +0.000, E1  +431.419, E3 -91459.915}
SPL {X  -124.554, Y  +771.914, Z    +0.000, E1  +430.935, E3 -91465.086}
SPL {X  -120.892, Y  +776.295, Z    +0.000, E1  +430.404, E3 -91469.969}
SPL {X  -118.039, Y  +779.498, Z    +0.000, E1  +429.949, E3 -91473.487}
SPL {X   -71.966, Y  +814.391, Z    +0.000, E1  +415.783, E3 -91612.140}
ENDSPLINE

SPLINE
SPL {X  -117.449, Y  +780.140, Z    +0.000, E1  +415.491, E3 -91776.554}
SPL {X  -137.837, Y  +752.727, Z    +0.000, E1  +411.385, E3 -91796.042}
SPL {X  -150.415, Y  +726.018, Z    +0.000, E1  +402.769, E3 -91804.917}
SPL {X  -156.153, Y  +706.328, Z    +0.000, E1  +392.414, E3 -91808.609}
SPL {X  -159.178, Y  +687.603, Z    +0.000, E1  +378.267, E3 -91810.587}
SPL {X  -159.915, Y  +676.399, Z    +0.000, E1  +367.484, E3 -91811.157}
SPL {X  -159.990, Y  +669.381, Z    +0.000, E1  +359.965, E3 -91811.257}
SPL {X  -159.990, Y  +666.412, Z    +0.000, E1  +352.765, E3 -91811.288}
SPL {X  -159.990, Y  +662.995, Z    +0.000, E1  +343.976, E3 -91811.391}
SPL {X  -159.990, Y  +658.179, Z    +0.000, E1  +331.312, E3 -91811.628}
SPL {X  -159.990, Y  +652.822, Z    +0.000, E1  +319.345, E3 -91812.042}
SPL {X  -159.990, Y  +646.185, Z    +0.000, E1  +308.728, E3 -91812.781}
SPL {X  -159.990, Y  +632.371, Z    +0.000, E1  +297.040, E3 -91815.134}
SPL {X  -159.990, Y  +579.000, Z    +0.000, E1  +286.931, E3 -91830.006}
SPL {X  -157.725, Y  +355.675, Z    +0.000, E1  +284.959, E3 -91926.964}
SPL {X  -142.593, Y  +309.947, Z    +0.000, E1  +282.426, E3 -91920.628}
SPL {X  -142.198, Y  +309.176, Z    +0.000, E1  +283.218, E3 -91929.436}
ENDSPLINE

SPLINE
SPL {X  -142.352, Y  +309.474, Z    +0.000, E1  +284.206, E3 -91939.130}
ENDSPLINE

SPLINE
SPL {X  -141.553, Y  +307.937, Z    +0.000, E1  +285.290, E3 -91950.146}
SPL {X  -140.562, Y  +306.086, Z    +0.000, E1  +286.440, E3 -91960.839}
SPL {X  -138.743, Y  +302.832, Z    +0.000, E1  +287.062, E3 -91967.637}
SPL {X  -135.531, Y  +297.482, Z    +0.000, E1  +287.444, E3 -91973.471}
SPL {X  -132.271, Y  +292.493, Z    +0.000, E1  +287.844, E3 -91978.990}
SPL {X  -128.837, Y  +287.643, Z    +0.000, E1  +288.283, E3 -91984.428}
SPL {X  -125.941, Y  +283.830, Z    +0.000, E1  +288.683, E3 -91988.727}
SPL {X  -122.669, Y  +279.791, Z    +0.000, E1  +289.119, E3 -91993.221}
SPL {X  -119.730, Y  +276.380, Z    +0.000, E1  +289.584, E3 -91997.009}
SPL {X   -74.058, Y  +240.683, Z    +0.000, E1  +305.011, E3 -92152.725}
ENDSPLINE

SPLINE
SPL {X  -130.401, Y  +289.805, Z    +0.000, E1  +307.505, E3 -92309.696}
SPL {X  -152.244, Y  +333.323, Z    +0.000, E1  +320.871, E3 -92326.508}
SPL {X  -158.218, Y  +358.753, Z    +0.000, E1  +336.397, E3 -92330.680}
SPL {X  -159.681, Y  +372.564, Z    +0.000, E1  +347.981, E3 -92331.731}
SPL {X  -159.987, Y  +381.561, Z    +0.000, E1  +356.806, E3 -92332.028}
SPL {X  -159.990, Y  +384.668, Z    +0.000, E1  +360.183, E3 -92332.054}
SPL {X  -159.990, Y  +387.837, Z    +0.000, E1  +367.342, E3 -92332.094}
SPL {X  -159.990, Y  +393.084, Z    +0.000, E1  +380.137, E3 -92332.304}
SPL {X  -159.990, Y  +401.914, Z    +0.000, E1  +400.147, E3 -92332.998}
SPL {X  -159.990, Y  +414.609, Z    +0.000, E1  +416.791, E3 -92334.735}
SPL {X  -159.990, Y  +464.476, Z    +0.000, E1  +431.765, E3 -92347.536}
SPL {X  -157.643, Y  +698.802, Z    +0.000, E1  +434.751, E3 -92450.550}
SPL {X  -154.470, Y  +713.164, Z    +0.000, E1  +434.425, E3 -92462.139}
SPL {X  -151.032, Y  +724.285, Z    +0.000, E1  +434.102, E3 -92471.943}
SPL {X  -147.134, Y  +734.337, Z    +0.000, E1  +433.686, E3 -92481.580}
SPL {X  -143.804, Y  +741.622, Z    +0.000, E1  +433.324, E3 -92488.968}
SPL {X  -140.603, Y  +747.839, Z    +0.000, E1  +432.964, E3 -92495.484}
SPL {X  -137.184, Y  +753.824, Z    +0.000, E1  +432.574, E3 -92501.920}
SPL {X  -133.762, Y  +759.276, Z    +0.000, E1  +432.150, E3 -92507.974}
SPL {X  -130.927, Y  +763.451, Z    +0.000, E1  +431.785, E3 -92512.669}
SPL {X  -126.852, Y  +768.996, Z    +0.000, E1  +431.276, E3 -92518.900}
SPL {X  -122.512, Y  +774.396, Z    +0.000, E1  +430.640, E3 -92525.009}
SPL {X  -119.782, Y  +777.562, Z    +0.000, E1  +430.221, E3 -92528.516}
SPL {X   -71.924, Y  +814.412, Z    +0.000, E1  +415.124, E3 -92685.386}
ENDSPLINE

SPLINE
SPL {X  -132.255, Y  +761.530, Z    +0.000, E1  +413.203, E3 -92848.556}
SPL {X  -150.415, Y  +726.018, Z    +0.000, E1  +402.769, E3 -92862.060}
SPL {X  -156.153, Y  +706.328, Z    +0.000, E1  +392.414, E3 -92865.752}
SPL {X  -159.178, Y  +687.603, Z    +0.000, E1  +378.267, E3 -92867.730}
SPL {X  -159.974, Y  +673.783, Z    +0.000, E1  +364.843, E3 -92868.352}
SPL {X  -159.990, Y  +669.500, Z    +0.000, E1  +360.000, E3 -92868.399}
SPL {X  -159.990, Y  +667.470, Z    +0.000, E1  +355.588, E3 -92868.417}
SPL {X  -159.990, Y  +662.995, Z    +0.000, E1  +343.976, E3 -92868.534}
SPL {X  -159.990, Y  +658.179, Z    +0.000, E1  +331.312, E3 -92868.770}
SPL {X  -159.990, Y  +652.822, Z    +0.000, E1  +319.345, E3 -92869.185}
SPL {X  -159.990, Y  +646.185, Z    +0.000, E1  +308.728, E3 -92869.924}
SPL {X  -159.990, Y  +632.371, Z    +0.000, E1  +297.040, E3 -92872.276}
SPL {X  -159.990, Y  +579.000, Z    +0.000, E1  +286.931, E3 -92887.149}
SPL {X  -157.725, Y  +355.675, Z    +0.000, E1  +284.959, E3 -92984.107}
SPL {X  -142.593, Y  +309.947, Z    +0.000, E1  +282.426, E3 -92977.770}
SPL {X  -142.198, Y  +309.176, Z    +0.000, E1  +283.218, E3 -92986.579}
ENDSPLINE

SPLINE
SPL {X  -142.352, Y  +309.474, Z    +0.000, E1  +284.206, E3 -92996.273}
ENDSPLINE

SPLINE
SPL {X  -141.553, Y  +307.937, Z    +0.000, E1  +285.290, E3 -93007.288}
SPL {X  -140.562, Y  +306.086, Z    +0.000, E1  +286.440, E3 -93017.982}
SPL {X  -138.743, Y  +302.832, Z    +0.000, E1  +287.062, E3 -93024.780}
SPL {X  -135.531, Y  +297.482, Z    +0.000, E1  +287.444, E3 -93030.614}
SPL {X  -132.271, Y  +292.493, Z    +0.000, E1  +287.844, E3 -93036.133}
SPL {X  -128.837, Y  +287.643, Z    +0.000, E1  +288.283, E3 -93041.570}
SPL {X  -124.965, Y  +282.598, Z    +0.000, E1  +288.800, E3 -93047.232}
SPL {X  -120.791, Y  +277.589, Z    +0.000, E1  +289.397, E3 -93052.805}
SPL {X   -74.058, Y  +240.683, Z    +0.000, E1  +305.011, E3 -93209.868}
ENDSPLINE

SPLINE
SPL {X  -130.401, Y  +289.805, Z    +0.000, E1  +307.505, E3 -93366.839}
SPL {X  -148.502, Y  +322.968, Z    +0.000, E1  +316.497, E3 -93381.159}
SPL {X  -154.800, Y  +342.080, Z    +0.000, E1  +325.471, E3 -93385.463}
SPL {X  -158.218, Y  +358.753, Z    +0.000, E1  +336.397, E3 -93387.823}
SPL {X  -159.681, Y  +372.564, Z    +0.000, E1  +347.981, E3 -93388.874}
SPL {X  -159.987, Y  +381.561, Z    +0.000, E1  +356.806, E3 -93389.171}
SPL {X  -159.990, Y  +384.668, Z    +0.000, E1  +360.183, E3 -93389.196}
SPL {X  -159.990, Y  +387.837, Z    +0.000, E1  +367.342, E3 -93389.237}
SPL {X  -159.990, Y  +393.084, Z    +0.000, E1  +380.137, E3 -93389.447}
SPL {X  -159.990, Y  +401.914, Z    +0.000, E1  +400.147, E3 -93390.141}
SPL {X  -159.990, Y  +414.609, Z    +0.000, E1  +416.791, E3 -93391.877}
SPL {X  -159.990, Y  +464.476, Z    +0.000, E1  +431.765, E3 -93404.678}
SPL {X  -157.643, Y  +698.802, Z    +0.000, E1  +434.751, E3 -93507.693}
SPL {X  -154.470, Y  +713.164, Z    +0.000, E1  +434.425, E3 -93519.282}
SPL {X  -151.032, Y  +724.285, Z    +0.000, E1  +434.102, E3 -93529.086}
SPL {X  -147.134, Y  +734.337, Z    +0.000, E1  +433.686, E3 -93538.723}
SPL {X  -143.804, Y  +741.622, Z    +0.000, E1  +433.324, E3 -93546.111}
SPL {X  -140.603, Y  +747.839, Z    +0.000, E1  +432.964, E3 -93552.627}
SPL {X  -137.184, Y  +753.824, Z    +0.000, E1  +432.574, E3 -93559.063}
SPL {X  -133.762, Y  +759.276, Z    +0.000, E1  +432.150, E3 -93565.117}
SPL {X  -130.927, Y  +763.451, Z    +0.000, E1  +431.785, E3 -93569.812}
SPL {X  -126.852, Y  +768.996, Z    +0.000, E1  +431.276, E3 -93576.042}
SPL {X  -122.512, Y  +774.396, Z    +0.000, E1  +430.640, E3 -93582.152}
SPL {X  -119.782, Y  +777.562, Z    +0.000, E1  +430.221, E3 -93585.659}
SPL {X   -71.924, Y  +814.412, Z    +0.000, E1  +415.124, E3 -93742.529}
ENDSPLINE

SPLINE
SPL {X  -132.255, Y  +761.530, Z    +0.000, E1  +413.203, E3 -93905.699}
SPL {X  -150.415, Y  +726.018, Z    +0.000, E1  +402.769, E3 -93919.203}
SPL {X  -156.153, Y  +706.328, Z    +0.000, E1  +392.414, E3 -93922.895}
SPL {X  -159.178, Y  +687.603, Z    +0.000, E1  +378.267, E3 -93924.873}
SPL {X  -159.974, Y  +673.783, Z    +0.000, E1  +364.843, E3 -93925.495}
SPL {X  -159.990, Y  +669.500, Z    +0.000, E1  +360.000, E3 -93925.542}
SPL {X  -159.990, Y  +667.470, Z    +0.000, E1  +355.588, E3 -93925.560}
SPL {X  -159.990, Y  +662.995, Z    +0.000, E1  +343.976, E3 -93925.677}
SPL {X  -159.990, Y  +658.179, Z    +0.000, E1  +331.312, E3 -93925.913}
SPL {X  -159.990, Y  +652.822, Z    +0.000, E1  +319.345, E3 -93926.328}
SPL {X  -159.990, Y  +646.185, Z    +0.000, E1  +308.728, E3 -93927.067}
SPL {X  -159.990, Y  +636.375, Z    +0.000, E1  +299.286, E3 -93928.506}
SPL {X  -159.990, Y  +617.374, Z    +0.000, E1  +291.478, E3 -93932.833}
SPL {X  -159.990, Y  +579.000, Z    +0.000, E1  +286.931, E3 -93944.292}
SPL {X  -157.725, Y  +355.675, Z    +0.000, E1  +284.959, E3 -94041.250}
SPL {X  -142.593, Y  +309.947, Z    +0.000, E1  +282.426, E3 -94034.913}
SPL {X  -142.198, Y  +309.176, Z    +0.000, E1  +283.218, E3 -94043.722}
ENDSPLINE

SPLINE
SPL {X  -142.352, Y  +309.474, Z    +0.000, E1  +284.206, E3 -94053.415}
ENDSPLINE

SPLINE
SPL {X  -141.929, Y  +308.657, Z    +0.000, E1  +285.131, E3 -94062.501}
SPL {X  -140.635, Y  +306.221, Z    +0.000, E1  +286.163, E3 -94072.913}
SPL {X  -138.743, Y  +302.832, Z    +0.000, E1  +287.062, E3 -94081.923}
SPL {X  -135.531, Y  +297.482, Z    +0.000, E1  +287.444, E3 -94087.757}
SPL {X  -132.271, Y  +292.493, Z    +0.000, E1  +287.844, E3 -94093.276}
SPL {X  -128.837, Y  +287.643, Z    +0.000, E1  +288.283, E3 -94098.713}
SPL {X  -125.941, Y  +283.830, Z    +0.000, E1  +288.683, E3 -94103.013}
SPL {X  -124.080, Y  +281.501, Z    +0.000, E1  +288.943, E3 -94105.624}
SPL {X  -120.791, Y  +277.589, Z    +0.000, E1  +289.397, E3 -94109.948}
SPL {X   -74.058, Y  +240.683, Z    +0.000, E1  +305.011, E3 -94267.011}
ENDSPLINE

SPLINE
SPL {X  -130.401, Y  +289.805, Z    +0.000, E1  +307.505, E3 -94423.982}
SPL {X  -152.244, Y  +333.323, Z    +0.000, E1  +320.871, E3 -94440.793}
SPL {X  -158.218, Y  +358.753, Z    +0.000, E1  +336.397, E3 -94444.966}
SPL {X  -159.681, Y  +372.564, Z    +0.000, E1  +347.981, E3 -94446.017}
SPL {X  -159.987, Y  +381.561, Z    +0.000, E1  +356.806, E3 -94446.314}
SPL {X  -159.990, Y  +384.668, Z    +0.000, E1  +360.183, E3 -94446.339}
SPL {X  -159.990, Y  +387.837, Z    +0.000, E1  +367.342, E3 -94446.380}
SPL {X  -159.990, Y  +393.084, Z    +0.000, E1  +380.137, E3 -94446.590}
SPL {X  -159.990, Y  +401.914, Z    +0.000, E1  +400.147, E3 -94447.283}
SPL {X  -159.990, Y  +414.609, Z    +0.000, E1  +416.791, E3 -94449.020}
SPL {X  -159.990, Y  +464.476, Z    +0.000, E1  +431.765, E3 -94461.821}
SPL {X  -157.643, Y  +698.802, Z    +0.000, E1  +434.751, E3 -94564.836}
SPL {X  -154.470, Y  +713.164, Z    +0.000, E1  +434.425, E3 -94576.425}
SPL {X  -152.098, Y  +721.129, Z    +0.000, E1  +434.190, E3 -94583.397}
SPL {X  -148.128, Y  +731.956, Z    +0.000, E1  +433.814, E3 -94593.478}
SPL {X  -143.804, Y  +741.622, Z    +0.000, E1  +433.324, E3 -94603.254}
SPL {X  -140.603, Y  +747.839, Z    +0.000, E1  +432.964, E3 -94609.769}
SPL {X  -137.184, Y  +753.824, Z    +0.000, E1  +432.574, E3 -94616.206}
SPL {X  -133.762, Y  +759.276, Z    +0.000, E1  +432.150, E3 -94622.260}
SPL {X  -130.927, Y  +763.451, Z    +0.000, E1  +431.785, E3 -94626.954}
SPL {X  -126.852, Y  +768.996, Z    +0.000, E1  +431.276, E3 -94633.185}
SPL {X  -122.512, Y  +774.396, Z    +0.000, E1  +430.640, E3 -94639.295}
SPL {X  -119.782, Y  +777.562, Z    +0.000, E1  +430.221, E3 -94642.802}
SPL {X   -71.924, Y  +814.412, Z    +0.000, E1  +415.124, E3 -94799.672}
ENDSPLINE

SPLINE
SPL {X  -132.255, Y  +761.530, Z    +0.000, E1  +413.203, E3 -94962.842}
SPL {X  -150.415, Y  +726.018, Z    +0.000, E1  +402.769, E3 -94976.346}
SPL {X  -157.206, Y  +701.216, Z    +0.000, E1  +389.056, E3 -94980.684}
SPL {X  -159.772, Y  +679.843, Z    +0.000, E1  +371.089, E3 -94982.448}
SPL {X  -159.990, Y  +669.585, Z    +0.000, E1  +360.185, E3 -94982.685}
SPL {X  -159.990, Y  +667.470, Z    +0.000, E1  +355.588, E3 -94982.703}
SPL {X  -159.990, Y  +662.995, Z    +0.000, E1  +343.976, E3 -94982.819}
SPL {X  -159.990, Y  +658.179, Z    +0.000, E1  +331.312, E3 -94983.056}
SPL {X  -159.990, Y  +652.822, Z    +0.000, E1  +319.345, E3 -94983.471}
SPL {X  -159.990, Y  +646.185, Z    +0.000, E1  +308.728, E3 -94984.210}
SPL {X  -159.990, Y  +632.371, Z    +0.000, E1  +297.040, E3 -94986.562}
SPL {X  -159.990, Y  +579.000, Z    +0.000, E1  +286.931, E3 -95001.434}
SPL {X  -157.725, Y  +355.675, Z    +0.000, E1  +284.959, E3 -95098.393}
SPL {X  -142.593, Y  +309.947, Z    +0.000, E1  +282.426, E3 -95092.056}
SPL {X  -142.198, Y  +309.176, Z    +0.000, E1  +283.218, E3 -95100.865}
ENDSPLINE

SPLINE
SPL {X  -142.352, Y  +309.474, Z    +0.000, E1  +284.206, E3 -95110.558}
ENDSPLINE

SPLINE
SPL {X  -141.929, Y  +308.657, Z    +0.000, E1  +285.131, E3 -95119.644}
SPL {X  -140.635, Y  +306.221, Z    +0.000, E1  +286.163, E3 -95130.056}
SPL {X  -138.743, Y  +302.832, Z    +0.000, E1  +287.062, E3 -95139.065}
SPL {X  -135.531, Y  +297.482, Z    +0.000, E1  +287.444, E3 -95144.900}
SPL {X  -132.271, Y  +292.493, Z    +0.000, E1  +287.844, E3 -95150.418}
SPL {X  -128.837, Y  +287.643, Z    +0.000, E1  +288.283, E3 -95155.856}
SPL {X  -124.965, Y  +282.598, Z    +0.000, E1  +288.800, E3 -95161.518}
SPL {X  -120.791, Y  +277.589, Z    +0.000, E1  +289.397, E3 -95167.091}
SPL {X   -74.058, Y  +240.683, Z    +0.000, E1  +305.011, E3 -95324.154}
ENDSPLINE

SPLINE
SPL {X  -130.401, Y  +289.805, Z    +0.000, E1  +307.505, E3 -95481.125}
SPL {X  -148.502, Y  +322.968, Z    +0.000, E1  +316.497, E3 -95495.445}
SPL {X  -154.800, Y  +342.080, Z    +0.000, E1  +325.471, E3 -95499.749}
SPL {X  -158.218, Y  +358.753, Z    +0.000, E1  +336.397, E3 -95502.108}
SPL {X  -159.681, Y  +372.564, Z    +0.000, E1  +347.981, E3 -95503.160}
SPL {X  -159.987, Y  +381.561, Z    +0.000, E1  +356.806, E3 -95503.456}
SPL {X  -159.990, Y  +384.668, Z    +0.000, E1  +360.183, E3 -95503.482}
SPL {X  -159.990, Y  +387.837, Z    +0.000, E1  +367.342, E3 -95503.523}
SPL {X  -159.990, Y  +393.084, Z    +0.000, E1  +380.137, E3 -95503.733}
SPL {X  -159.990, Y  +401.914, Z    +0.000, E1  +400.147, E3 -95504.426}
SPL {X  -159.990, Y  +414.609, Z    +0.000, E1  +416.791, E3 -95506.163}
SPL {X  -159.990, Y  +464.476, Z    +0.000, E1  +431.765, E3 -95518.964}
SPL {X  -157.643, Y  +698.802, Z    +0.000, E1  +434.751, E3 -95621.979}
SPL {X  -154.470, Y  +713.164, Z    +0.000, E1  +434.425, E3 -95633.568}
SPL {X  -151.032, Y  +724.285, Z    +0.000, E1  +434.102, E3 -95643.371}
SPL {X  -147.134, Y  +734.337, Z    +0.000, E1  +433.686, E3 -95653.009}
SPL {X  -143.804, Y  +741.622, Z    +0.000, E1  +433.324, E3 -95660.397}
SPL {X  -140.603, Y  +747.839, Z    +0.000, E1  +432.964, E3 -95666.912}
SPL {X  -137.184, Y  +753.824, Z    +0.000, E1  +432.574, E3 -95673.349}
SPL {X  -133.762, Y  +759.276, Z    +0.000, E1  +432.150, E3 -95679.403}
SPL {X  -130.927, Y  +763.451, Z    +0.000, E1  +431.785, E3 -95684.097}
SPL {X  -128.105, Y  +767.343, Z    +0.000, E1  +431.419, E3 -95688.486}
SPL {X  -124.554, Y  +771.914, Z    +0.000, E1  +430.935, E3 -95693.657}
SPL {X  -120.892, Y  +776.295, Z    +0.000, E1  +430.404, E3 -95698.541}
SPL {X  -118.039, Y  +779.498, Z    +0.000, E1  +429.949, E3 -95702.059}
SPL {X   -71.924, Y  +814.412, Z    +0.000, E1  +415.124, E3 -95856.815}
ENDSPLINE

SPLINE
SPL {X  -132.255, Y  +761.530, Z    +0.000, E1  +413.203, E3 -96019.984}
SPL {X  -150.415, Y  +726.018, Z    +0.000, E1  +402.769, E3 -96033.488}
SPL {X  -156.153, Y  +706.328, Z    +0.000, E1  +392.414, E3 -96037.181}
SPL {X  -159.178, Y  +687.603, Z    +0.000, E1  +378.267, E3 -96039.158}
SPL {X  -159.974, Y  +673.783, Z    +0.000, E1  +364.843, E3 -96039.780}
SPL {X  -159.990, Y  +669.500, Z    +0.000, E1  +360.000, E3 -96039.828}
SPL {X  -159.990, Y  +667.470, Z    +0.000, E1  +355.588, E3 -96039.846}
SPL {X  -159.990, Y  +662.995, Z    +0.000, E1  +343.976, E3 -96039.962}
SPL {X  -159.990, Y  +658.179, Z    +0.000, E1  +331.312, E3 -96040.199}
SPL {X  -159.990, Y  +652.822, Z    +0.000, E1  +319.345, E3 -96040.614}
SPL {X  -159.990, Y  +646.185, Z    +0.000, E1  +308.728, E3 -96041.352}
SPL {X  -159.990, Y  +636.375, Z    +0.000, E1  +299.286, E3 -96042.792}
SPL {X  -159.990, Y  +617.374, Z    +0.000, E1  +291.478, E3 -96047.118}
SPL {X  -159.990, Y  +579.000, Z    +0.000, E1  +286.931, E3 -96058.577}
SPL {X  -157.725, Y  +355.675, Z    +0.000, E1  +284.959, E3 -96155.536}
SPL {X  -142.593, Y  +309.947, Z    +0.000, E1  +282.426, E3 -96149.199}
SPL {X  -142.198, Y  +309.176, Z    +0.000, E1  +283.218, E3 -96158.008}
ENDSPLINE

SPLINE
SPL {X  -142.352, Y  +309.474, Z    +0.000, E1  +284.206, E3 -96167.701}
ENDSPLINE

SPLINE
SPL {X  -141.553, Y  +307.937, Z    +0.000, E1  +285.290, E3 -96178.717}
SPL {X  -140.562, Y  +306.086, Z    +0.000, E1  +286.440, E3 -96189.411}
SPL {X  -138.743, Y  +302.832, Z    +0.000, E1  +287.062, E3 -96196.208}
SPL {X  -135.531, Y  +297.482, Z    +0.000, E1  +287.444, E3 -96202.043}
SPL {X  -132.271, Y  +292.493, Z    +0.000, E1  +287.844, E3 -96207.561}
SPL {X  -128.837, Y  +287.643, Z    +0.000, E1  +288.283, E3 -96212.999}
SPL {X  -124.965, Y  +282.598, Z    +0.000, E1  +288.800, E3 -96218.661}
SPL {X  -120.791, Y  +277.589, Z    +0.000, E1  +289.397, E3 -96224.234}
SPL {X   -74.058, Y  +240.683, Z    +0.000, E1  +305.011, E3 -96381.297}
ENDSPLINE

SPLINE
SPL {X  -130.401, Y  +289.805, Z    +0.000, E1  +307.505, E3 -96538.267}
SPL {X  -148.502, Y  +322.968, Z    +0.000, E1  +316.497, E3 -96552.588}
SPL {X  -154.800, Y  +342.080, Z    +0.000, E1  +325.471, E3 -96556.891}
SPL {X  -158.218, Y  +358.753, Z    +0.000, E1  +336.397, E3 -96559.251}
SPL {X  -159.681, Y  +372.564, Z    +0.000, E1  +347.981, E3 -96560.303}
SPL {X  -159.987, Y  +381.561, Z    +0.000, E1  +356.806, E3 -96560.599}
SPL {X  -159.990, Y  +384.668, Z    +0.000, E1  +360.183, E3 -96560.625}
SPL {X  -159.990, Y  +387.837, Z    +0.000, E1  +367.342, E3 -96560.666}
SPL {X  -159.990, Y  +393.084, Z    +0.000, E1  +380.137, E3 -96560.876}
SPL {X  -159.990, Y  +401.914, Z    +0.000, E1  +400.147, E3 -96561.569}
SPL {X  -159.990, Y  +414.609, Z    +0.000, E1  +416.791, E3 -96563.306}
SPL {X  -159.990, Y  +464.476, Z    +0.000, E1  +431.765, E3 -96576.107}
SPL {X  -157.643, Y  +698.802, Z    +0.000, E1  +434.751, E3 -96679.122}
SPL {X  -154.470, Y  +713.164, Z    +0.000, E1  +434.425, E3 -96690.710}
SPL {X  -152.098, Y  +721.129, Z    +0.000, E1  +434.190, E3 -96697.683}
SPL {X  -148.128, Y  +731.956, Z    +0.000, E1  +433.814, E3 -96707.763}
SPL {X  -143.804, Y  +741.622, Z    +0.000, E1  +433.324, E3 -96717.540}
SPL {X  -140.603, Y  +747.839, Z    +0.000, E1  +432.964, E3 -96724.055}
SPL {X  -137.184, Y  +753.824, Z    +0.000, E1  +432.574, E3 -96730.492}
SPL {X  -133.762, Y  +759.276, Z    +0.000, E1  +432.150, E3 -96736.546}
SPL {X  -130.927, Y  +763.451, Z    +0.000, E1  +431.785, E3 -96741.240}
SPL {X  -126.852, Y  +768.996, Z    +0.000, E1  +431.276, E3 -96747.471}
SPL {X  -122.512, Y  +774.396, Z    +0.000, E1  +430.640, E3 -96753.580}
SPL {X  -119.782, Y  +777.562, Z    +0.000, E1  +430.221, E3 -96757.088}
SPL {X   -71.966, Y  +814.391, Z    +0.000, E1  +415.783, E3 -96897.854}
ENDSPLINE

SPLINE
SPL {X  -117.449, Y  +780.140, Z    +0.000, E1  +415.491, E3 -97062.268}
SPL {X  -137.837, Y  +752.727, Z    +0.000, E1  +411.385, E3 -97081.756}
SPL {X  -150.415, Y  +726.018, Z    +0.000, E1  +402.769, E3 -97090.631}
SPL {X  -156.153, Y  +706.328, Z    +0.000, E1  +392.414, E3 -97094.323}
SPL {X  -159.178, Y  +687.603, Z    +0.000, E1  +378.267, E3 -97096.301}
SPL {X  -159.974, Y  +673.783, Z    +0.000, E1  +364.843, E3 -97096.923}
SPL {X  -159.990, Y  +669.500, Z    +0.000, E1  +360.000, E3 -97096.971}
SPL {X  -159.990, Y  +667.470, Z    +0.000, E1  +355.588, E3 -97096.989}
SPL {X  -159.990, Y  +662.995, Z    +0.000, E1  +343.976, E3 -97097.105}
SPL {X  -159.990, Y  +658.179, Z    +0.000, E1  +331.312, E3 -97097.342}
SPL {X  -159.990, Y  +652.822, Z    +0.000, E1  +319.345, E3 -97097.757}
SPL {X  -159.990, Y  +646.185, Z    +0.000, E1  +308.728, E3 -97098.495}
SPL {X  -159.990, Y  +636.375, Z    +0.000, E1  +299.286, E3 -97099.935}
SPL {X  -159.990, Y  +617.374, Z    +0.000, E1  +291.478, E3 -97104.261}
SPL {X  -159.990, Y  +579.000, Z    +0.000, E1  +286.931, E3 -97115.720}
SPL {X  -157.725, Y  +355.675, Z    +0.000, E1  +284.959, E3 -97212.678}
SPL {X  -142.593, Y  +309.947, Z    +0.000, E1  +282.426, E3 -97206.342}
SPL {X  -142.198, Y  +309.176, Z    +0.000, E1  +283.218, E3 -97215.150}
ENDSPLINE

SPLINE
SPL {X  -142.352, Y  +309.474, Z    +0.000, E1  +284.206, E3 -97224.844}
ENDSPLINE

SPLINE
SPL {X  -141.553, Y  +307.937, Z    +0.000, E1  +285.290, E3 -97235.860}
SPL {X  -140.562, Y  +306.086, Z    +0.000, E1  +286.440, E3 -97246.554}
SPL {X  -138.743, Y  +302.832, Z    +0.000, E1  +287.062, E3 -97253.351}
SPL {X  -135.531, Y  +297.482, Z    +0.000, E1  +287.444, E3 -97259.186}
SPL {X  -132.271, Y  +292.493, Z    +0.000, E1  +287.844, E3 -97264.704}
SPL {X  -128.837, Y  +287.643, Z    +0.000, E1  +288.283, E3 -97270.142}
SPL {X  -124.965, Y  +282.598, Z    +0.000, E1  +288.800, E3 -97275.804}
SPL {X  -120.791, Y  +277.589, Z    +0.000, E1  +289.397, E3 -97281.376}
SPL {X   -74.058, Y  +240.683, Z    +0.000, E1  +305.011, E3 -97438.439}
ENDSPLINE

SPLINE
SPL {X  -130.401, Y  +289.805, Z    +0.000, E1  +307.505, E3 -97595.410}
SPL {X  -148.502, Y  +322.968, Z    +0.000, E1  +316.497, E3 -97609.731}
SPL {X  -154.800, Y  +342.080, Z    +0.000, E1  +325.471, E3 -97614.034}
SPL {X  -158.218, Y  +358.753, Z    +0.000, E1  +336.397, E3 -97616.394}
SPL {X  -159.681, Y  +372.564, Z    +0.000, E1  +347.981, E3 -97617.446}
SPL {X  -159.987, Y  +381.561, Z    +0.000, E1  +356.806, E3 -97617.742}
SPL {X  -159.990, Y  +384.668, Z    +0.000, E1  +360.183, E3 -97617.768}
SPL {X  -159.990, Y  +389.080, Z    +0.000, E1  +370.094, E3 -97617.848}
SPL {X  -159.990, Y  +394.652, Z    +0.000, E1  +384.399, E3 -97618.097}
SPL {X  -159.990, Y  +401.914, Z    +0.000, E1  +400.147, E3 -97618.712}
SPL {X  -159.990, Y  +414.609, Z    +0.000, E1  +416.791, E3 -97620.449}
SPL {X  -159.990, Y  +464.476, Z    +0.000, E1  +431.765, E3 -97633.250}
SPL {X  -157.643, Y  +698.802, Z    +0.000, E1  +434.751, E3 -97736.265}
SPL {X  -154.470, Y  +713.164, Z    +0.000, E1  +434.425, E3 -97747.853}
SPL {X  -151.032, Y  +724.285, Z    +0.000, E1  +434.102, E3 -97757.657}
SPL {X  -147.134, Y  +734.337, Z    +0.000, E1  +433.686, E3 -97767.295}
SPL {X  -143.804, Y  +741.622, Z    +0.000, E1  +433.324, E3 -97774.682}
SPL {X  -140.603, Y  +747.839, Z    +0.000, E1  +432.964, E3 -97781.198}
SPL {X  -137.184, Y  +753.824, Z    +0.000, E1  +432.574, E3 -97787.635}
SPL {X  -133.762, Y  +759.276, Z    +0.000, E1  +432.150, E3 -97793.688}
SPL {X  -130.927, Y  +763.451, Z    +0.000, E1  +431.785, E3 -97798.383}
SPL {X  -126.852, Y  +768.996, Z    +0.000, E1  +431.276, E3 -97804.614}
SPL {X  -122.512, Y  +774.396, Z    +0.000, E1  +430.640, E3 -97810.723}
SPL {X  -119.782, Y  +777.562, Z    +0.000, E1  +430.221, E3 -97814.230}
SPL {X   -71.966, Y  +814.391, Z    +0.000, E1  +415.783, E3 -97954.997}
ENDSPLINE

SPLINE
SPL {X  -117.449, Y  +780.140, Z    +0.000, E1  +415.491, E3 -98119.411}
SPL {X  -137.837, Y  +752.727, Z    +0.000, E1  +411.385, E3 -98138.899}
SPL {X  -150.415, Y  +726.018, Z    +0.000, E1  +402.769, E3 -98147.774}
SPL {X  -156.153, Y  +706.328, Z    +0.000, E1  +392.414, E3 -98151.466}
SPL {X  -159.178, Y  +687.603, Z    +0.000, E1  +378.267, E3 -98153.444}
SPL {X  -159.974, Y  +673.783, Z    +0.000, E1  +364.843, E3 -98154.066}
SPL {X  -159.990, Y  +669.500, Z    +0.000, E1  +360.000, E3 -98154.114}
SPL {X  -159.990, Y  +667.470, Z    +0.000, E1  +355.588, E3 -98154.132}
SPL {X  -159.990, Y  +662.995, Z    +0.000, E1  +343.976, E3 -98154.248}
SPL {X  -159.990, Y  +658.179, Z    +0.000, E1  +331.312, E3 -98154.485}
SPL {X  -159.990, Y  +652.822, Z    +0.000, E1  +319.345, E3 -98154.899}
SPL {X  -159.990, Y  +646.185, Z    +0.000, E1  +308.728, E3 -98155.638}
SPL {X  -159.990, Y  +632.371, Z    +0.000, E1  +297.040, E3 -98157.991}
SPL {X  -159.990, Y  +579.000, Z    +0.000, E1  +286.931, E3 -98172.863}
SPL {X  -157.725, Y  +355.675, Z    +0.000, E1  +284.959, E3 -98269.821}
SPL {X  -142.593, Y  +309.947, Z    +0.000, E1  +282.426, E3 -98263.485}
SPL {X  -142.198, Y  +309.176, Z    +0.000, E1  +283.218, E3 -98272.293}
ENDSPLINE

SPLINE
SPL {X  -142.352, Y  +309.474, Z    +0.000, E1  +284.206, E3 -98281.987}
ENDSPLINE

SPLINE
SPL {X  -141.553, Y  +307.937, Z    +0.000, E1  +285.290, E3 -98293.003}
SPL {X  -140.562, Y  +306.086, Z    +0.000, E1  +286.440, E3 -98303.697}
SPL {X  -138.743, Y  +302.832, Z    +0.000, E1  +287.062, E3 -98310.494}
SPL {X  -135.531, Y  +297.482, Z    +0.000, E1  +287.444, E3 -98316.329}
SPL {X  -132.271, Y  +292.493, Z    +0.000, E1  +287.844, E3 -98321.847}
SPL {X  -128.837, Y  +287.643, Z    +0.000, E1  +288.283, E3 -98327.285}
SPL {X  -124.965, Y  +282.598, Z    +0.000, E1  +288.800, E3 -98332.946}
SPL {X  -120.791, Y  +277.589, Z    +0.000, E1  +289.397, E3 -98338.519}
SPL {X   -74.058, Y  +240.683, Z    +0.000, E1  +305.011, E3 -98495.582}
ENDSPLINE

SPLINE
SPL {X  -130.401, Y  +289.805, Z    +0.000, E1  +307.505, E3 -98652.553}
SPL {X  -152.244, Y  +333.323, Z    +0.000, E1  +320.871, E3 -98669.365}
SPL {X  -158.218, Y  +358.753, Z    +0.000, E1  +336.397, E3 -98673.537}
SPL {X  -159.681, Y  +372.564, Z    +0.000, E1  +347.981, E3 -98674.589}
SPL {X  -159.987, Y  +381.561, Z    +0.000, E1  +356.806, E3 -98674.885}
SPL {X  -159.990, Y  +384.668, Z    +0.000, E1  +360.183, E3 -98674.911}
SPL {X  -159.990, Y  +387.837, Z    +0.000, E1  +367.342, E3 -98674.951}
SPL {X  -159.990, Y  +393.084, Z    +0.000, E1  +380.137, E3 -98675.161}
SPL {X  -159.990, Y  +401.914, Z    +0.000, E1  +400.147, E3 -98675.855}
SPL {X  -159.990, Y  +414.609, Z    +0.000, E1  +416.791, E3 -98677.592}
SPL {X  -159.990, Y  +464.476, Z    +0.000, E1  +431.765, E3 -98690.393}
SPL {X  -157.643, Y  +698.802, Z    +0.000, E1  +434.751, E3 -98793.407}
SPL {X  -154.470, Y  +713.164, Z    +0.000, E1  +434.425, E3 -98804.996}
SPL {X  -152.098, Y  +721.129, Z    +0.000, E1  +434.190, E3 -98811.968}
SPL {X  -148.128, Y  +731.956, Z    +0.000, E1  +433.814, E3 -98822.049}
SPL {X  -143.804, Y  +741.622, Z    +0.000, E1  +433.324, E3 -98831.825}
SPL {X  -140.603, Y  +747.839, Z    +0.000, E1  +432.964, E3 -98838.341}
SPL {X  -137.184, Y  +753.824, Z    +0.000, E1  +432.574, E3 -98844.778}
SPL {X  -133.762, Y  +759.276, Z    +0.000, E1  +432.150, E3 -98850.831}
SPL {X  -130.927, Y  +763.451, Z    +0.000, E1  +431.785, E3 -98855.526}
SPL {X  -126.852, Y  +768.996, Z    +0.000, E1  +431.276, E3 -98861.757}
SPL {X  -122.512, Y  +774.396, Z    +0.000, E1  +430.640, E3 -98867.866}
SPL {X  -119.782, Y  +777.562, Z    +0.000, E1  +430.221, E3 -98871.373}
SPL {X   -71.924, Y  +814.412, Z    +0.000, E1  +415.124, E3 -99028.243}
ENDSPLINE

SPLINE
SPL {X  -132.255, Y  +761.530, Z    +0.000, E1  +413.203, E3 -99191.413}
SPL {X  -150.415, Y  +726.018, Z    +0.000, E1  +402.769, E3 -99204.917}
SPL {X  -156.153, Y  +706.328, Z    +0.000, E1  +392.414, E3 -99208.609}
SPL {X  -159.178, Y  +687.603, Z    +0.000, E1  +378.267, E3 -99210.587}
SPL {X  -159.974, Y  +673.783, Z    +0.000, E1  +364.843, E3 -99211.209}
SPL {X  -159.990, Y  +669.500, Z    +0.000, E1  +360.000, E3 -99211.256}
SPL {X  -159.990, Y  +667.470, Z    +0.000, E1  +355.588, E3 -99211.274}
SPL {X  -159.990, Y  +662.995, Z    +0.000, E1  +343.976, E3 -99211.391}
SPL {X  -159.990, Y  +658.179, Z    +0.000, E1  +331.312, E3 -99211.628}
SPL {X  -159.990, Y  +652.822, Z    +0.000, E1  +319.345, E3 -99212.042}
SPL {X  -159.990, Y  +646.185, Z    +0.000, E1  +308.728, E3 -99212.781}
SPL {X  -159.990, Y  +636.375, Z    +0.000, E1  +299.286, E3 -99214.220}
SPL {X  -159.990, Y  +617.374, Z    +0.000, E1  +291.478, E3 -99218.547}
SPL {X  -159.990, Y  +579.000, Z    +0.000, E1  +286.931, E3 -99230.006}
SPL {X  -157.725, Y  +355.675, Z    +0.000, E1  +284.959, E3 -99326.964}
SPL {X  -142.593, Y  +309.947, Z    +0.000, E1  +282.426, E3 -99320.628}
SPL {X  -142.198, Y  +309.176, Z    +0.000, E1  +283.218, E3 -99329.436}
ENDSPLINE

SPLINE
SPL {X  -142.352, Y  +309.474, Z    +0.000, E1  +284.206, E3 -99339.130}
ENDSPLINE

SPLINE
SPL {X  -141.929, Y  +308.657, Z    +0.000, E1  +285.131, E3 -99348.215}
SPL {X  -140.635, Y  +306.221, Z    +0.000, E1  +286.163, E3 -99358.627}
SPL {X  -138.743, Y  +302.832, Z    +0.000, E1  +287.062, E3 -99367.637}
SPL {X  -135.531, Y  +297.482, Z    +0.000, E1  +287.444, E3 -99373.471}
SPL {X  -132.271, Y  +292.493, Z    +0.000, E1  +287.844, E3 -99378.990}
SPL {X  -128.837, Y  +287.643, Z    +0.000, E1  +288.283, E3 -99384.428}
SPL {X  -125.941, Y  +283.830, Z    +0.000, E1  +288.683, E3 -99388.727}
SPL {X  -124.080, Y  +281.501, Z    +0.000, E1  +288.943, E3 -99391.338}
SPL {X  -120.791, Y  +277.589, Z    +0.000, E1  +289.397, E3 -99395.662}
SPL {X   -74.058, Y  +240.683, Z    +0.000, E1  +305.011, E3 -99552.725}
ENDSPLINE

SPLINE
SPL {X  -130.401, Y  +289.805, Z    +0.000, E1  +307.505, E3 -99709.696}
SPL {X  -152.244, Y  +333.323, Z    +0.000, E1  +320.871, E3 -99726.508}
SPL {X  -158.218, Y  +358.753, Z    +0.000, E1  +336.397, E3 -99730.680}
SPL {X  -159.681, Y  +372.564, Z    +0.000, E1  +347.981, E3 -99731.731}
SPL {X  -159.987, Y  +381.561, Z    +0.000, E1  +356.806, E3 -99732.028}
SPL {X  -159.990, Y  +384.668, Z    +0.000, E1  +360.183, E3 -99732.054}
SPL {X  -159.990, Y  +387.837, Z    +0.000, E1  +367.342, E3 -99732.094}
SPL {X  -159.990, Y  +393.084, Z    +0.000, E1  +380.137, E3 -99732.304}
SPL {X  -159.990, Y  +401.914, Z    +0.000, E1  +400.147, E3 -99732.998}
SPL {X  -159.990, Y  +414.609, Z    +0.000, E1  +416.791, E3 -99734.735}
SPL {X  -159.990, Y  +464.476, Z    +0.000, E1  +431.765, E3 -99747.536}
SPL {X  -157.643, Y  +698.802, Z    +0.000, E1  +434.751, E3 -99850.550}
SPL {X  -154.470, Y  +713.164, Z    +0.000, E1  +434.425, E3 -99862.139}
SPL {X  -152.098, Y  +721.129, Z    +0.000, E1  +434.190, E3 -99869.111}
SPL {X  -148.128, Y  +731.956, Z    +0.000, E1  +433.814, E3 -99879.192}
SPL {X  -143.804, Y  +741.622, Z    +0.000, E1  +433.324, E3 -99888.968}
SPL {X  -140.603, Y  +747.839, Z    +0.000, E1  +432.964, E3 -99895.484}
SPL {X  -137.184, Y  +753.824, Z    +0.000, E1  +432.574, E3 -99901.920}
SPL {X  -133.762, Y  +759.276, Z    +0.000, E1  +432.150, E3 -99907.974}
SPL {X  -130.927, Y  +763.451, Z    +0.000, E1  +431.785, E3 -99912.669}
SPL {X  -128.105, Y  +767.343, Z    +0.000, E1  +431.419, E3 -99917.058}
SPL {X  -125.461, Y  +770.778, Z    +0.000, E1  +431.046, E3 -99920.971}
SPL {X  -122.512, Y  +774.396, Z    +0.000, E1  +430.640, E3 -99925.009}
SPL {X  -119.782, Y  +777.562, Z    +0.000, E1  +430.221, E3 -99928.516}
SPL {X   -71.924, Y  +814.412, Z    +0.000, E1  +415.124, E3 -100085.386}
ENDSPLINE

SPLINE
SPL {X  -132.255, Y  +761.530, Z    +0.000, E1  +413.203, E3 -100248.556}
SPL {X  -150.415, Y  +726.018, Z    +0.000, E1  +402.769, E3 -100262.060}
SPL {X  -156.153, Y  +706.328, Z    +0.000, E1  +392.414, E3 -100265.752}
SPL {X  -159.178, Y  +687.603, Z    +0.000, E1  +378.267, E3 -100267.730}
SPL {X  -159.915, Y  +676.399, Z    +0.000, E1  +367.484, E3 -100268.300}
SPL {X  -159.990, Y  +669.585, Z    +0.000, E1  +360.185, E3 -100268.399}
SPL {X  -159.990, Y  +667.470, Z    +0.000, E1  +355.588, E3 -100268.417}
SPL {X  -159.990, Y  +662.995, Z    +0.000, E1  +343.976, E3 -100268.534}
SPL {X  -159.990, Y  +658.179, Z    +0.000, E1  +331.312, E3 -100268.770}
SPL {X  -159.990, Y  +652.822, Z    +0.000, E1  +319.345, E3 -100269.185}
SPL {X  -159.990, Y  +646.185, Z    +0.000, E1  +308.728, E3 -100269.924}
SPL {X  -159.990, Y  +636.375, Z    +0.000, E1  +299.286, E3 -100271.363}
SPL {X  -159.990, Y  +617.374, Z    +0.000, E1  +291.478, E3 -100275.690}
SPL {X  -159.990, Y  +579.000, Z    +0.000, E1  +286.931, E3 -100287.149}
SPL {X  -157.725, Y  +355.675, Z    +0.000, E1  +284.959, E3 -100384.107}
SPL {X  -142.593, Y  +309.947, Z    +0.000, E1  +282.426, E3 -100377.770}
SPL {X  -142.198, Y  +309.176, Z    +0.000, E1  +283.218, E3 -100386.579}
ENDSPLINE

SPLINE
SPL {X  -142.352, Y  +309.474, Z    +0.000, E1  +284.206, E3 -100396.273}
ENDSPLINE

SPLINE
SPL {X  -141.929, Y  +308.657, Z    +0.000, E1  +285.131, E3 -100405.358}
SPL {X  -140.635, Y  +306.221, Z    +0.000, E1  +286.163, E3 -100415.770}
SPL {X  -138.743, Y  +302.832, Z    +0.000, E1  +287.062, E3 -100424.780}
SPL {X  -135.531, Y  +297.482, Z    +0.000, E1  +287.444, E3 -100430.614}
SPL {X  -132.271, Y  +292.493, Z    +0.000, E1  +287.844, E3 -100436.133}
SPL {X  -128.837, Y  +287.643, Z    +0.000, E1  +288.283, E3 -100441.570}
SPL {X  -125.941, Y  +283.830, Z    +0.000, E1  +288.683, E3 -100445.870}
SPL {X  -124.080, Y  +281.501, Z    +0.000, E1  +288.943, E3 -100448.481}
SPL {X  -120.791, Y  +277.589, Z    +0.000, E1  +289.397, E3 -100452.805}
SPL {X   -74.058, Y  +240.683, Z    +0.000, E1  +305.011, E3 -100609.868}
ENDSPLINE

SPLINE
SPL {X  -130.401, Y  +289.805, Z    +0.000, E1  +307.505, E3 -100766.839}
SPL {X  -152.244, Y  +333.323, Z    +0.000, E1  +320.871, E3 -100783.650}
SPL {X  -158.218, Y  +358.753, Z    +0.000, E1  +336.397, E3 -100787.823}
SPL {X  -159.681, Y  +372.564, Z    +0.000, E1  +347.981, E3 -100788.874}
SPL {X  -159.987, Y  +381.561, Z    +0.000, E1  +356.806, E3 -100789.171}
SPL {X  -159.990, Y  +384.668, Z    +0.000, E1  +360.183, E3 -100789.196}
SPL {X  -159.990, Y  +387.837, Z    +0.000, E1  +367.342, E3 -100789.237}
SPL {X  -159.990, Y  +393.084, Z    +0.000, E1  +380.137, E3 -100789.447}
SPL {X  -159.990, Y  +401.914, Z    +0.000, E1  +400.147, E3 -100790.141}
SPL {X  -159.990, Y  +414.609, Z    +0.000, E1  +416.791, E3 -100791.877}
SPL {X  -159.990, Y  +464.476, Z    +0.000, E1  +431.765, E3 -100804.678}
SPL {X  -157.643, Y  +698.802, Z    +0.000, E1  +434.751, E3 -100907.693}
SPL {X  -154.470, Y  +713.164, Z    +0.000, E1  +434.425, E3 -100919.282}
SPL {X  -152.098, Y  +721.129, Z    +0.000, E1  +434.190, E3 -100926.254}
SPL {X  -148.128, Y  +731.956, Z    +0.000, E1  +433.814, E3 -100936.335}
SPL {X  -143.804, Y  +741.622, Z    +0.000, E1  +433.324, E3 -100946.111}
SPL {X  -140.603, Y  +747.839, Z    +0.000, E1  +432.964, E3 -100952.627}
SPL {X  -137.184, Y  +753.824, Z    +0.000, E1  +432.574, E3 -100959.063}
SPL {X  -133.762, Y  +759.276, Z    +0.000, E1  +432.150, E3 -100965.117}
SPL {X  -130.927, Y  +763.451, Z    +0.000, E1  +431.785, E3 -100969.812}
SPL {X  -126.852, Y  +768.996, Z    +0.000, E1  +431.276, E3 -100976.042}
SPL {X  -122.512, Y  +774.396, Z    +0.000, E1  +430.640, E3 -100982.152}
SPL {X  -119.782, Y  +777.562, Z    +0.000, E1  +430.221, E3 -100985.659}
SPL {X   -71.924, Y  +814.412, Z    +0.000, E1  +415.124, E3 -101142.529}
ENDSPLINE

SPLINE
SPL {X  -132.255, Y  +761.530, Z    +0.000, E1  +413.203, E3 -101305.699}
SPL {X  -150.415, Y  +726.018, Z    +0.000, E1  +402.769, E3 -101319.203}
SPL {X  -156.153, Y  +706.328, Z    +0.000, E1  +392.414, E3 -101322.895}
SPL {X  -159.178, Y  +687.603, Z    +0.000, E1  +378.267, E3 -101324.873}
SPL {X  -159.974, Y  +673.783, Z    +0.000, E1  +364.843, E3 -101325.495}
SPL {X  -159.990, Y  +669.500, Z    +0.000, E1  +360.000, E3 -101325.542}
SPL {X  -159.990, Y  +667.470, Z    +0.000, E1  +355.588, E3 -101325.560}
SPL {X  -159.990, Y  +662.995, Z    +0.000, E1  +343.976, E3 -101325.677}
SPL {X  -159.990, Y  +658.179, Z    +0.000, E1  +331.312, E3 -101325.913}
SPL {X  -159.990, Y  +652.822, Z    +0.000, E1  +319.345, E3 -101326.328}
SPL {X  -159.990, Y  +646.185, Z    +0.000, E1  +308.728, E3 -101327.067}
SPL {X  -159.990, Y  +636.375, Z    +0.000, E1  +299.286, E3 -101328.506}
SPL {X  -159.990, Y  +617.374, Z    +0.000, E1  +291.478, E3 -101332.833}
SPL {X  -159.990, Y  +579.000, Z    +0.000, E1  +286.931, E3 -101344.292}
SPL {X  -157.725, Y  +355.675, Z    +0.000, E1  +284.959, E3 -101441.250}
SPL {X  -142.593, Y  +309.947, Z    +0.000, E1  +282.426, E3 -101434.913}
SPL {X  -142.198, Y  +309.176, Z    +0.000, E1  +283.218, E3 -101443.722}
ENDSPLINE

SPLINE
SPL {X  -142.352, Y  +309.474, Z    +0.000, E1  +284.206, E3 -101453.415}
ENDSPLINE

SPLINE
SPL {X  -141.929, Y  +308.657, Z    +0.000, E1  +285.131, E3 -101462.501}
SPL {X  -140.635, Y  +306.221, Z    +0.000, E1  +286.163, E3 -101472.913}
SPL {X  -138.743, Y  +302.832, Z    +0.000, E1  +287.062, E3 -101481.923}
SPL {X  -135.531, Y  +297.482, Z    +0.000, E1  +287.444, E3 -101487.757}
SPL {X  -132.271, Y  +292.493, Z    +0.000, E1  +287.844, E3 -101493.276}
SPL {X  -128.837, Y  +287.643, Z    +0.000, E1  +288.283, E3 -101498.713}
SPL {X  -125.941, Y  +283.830, Z    +0.000, E1  +288.683, E3 -101503.013}
SPL {X  -124.080, Y  +281.501, Z    +0.000, E1  +288.943, E3 -101505.624}
SPL {X  -120.791, Y  +277.589, Z    +0.000, E1  +289.397, E3 -101509.948}
SPL {X   -74.058, Y  +240.683, Z    +0.000, E1  +305.011, E3 -101667.011}
ENDSPLINE

SPLINE
SPL {X  -130.401, Y  +289.805, Z    +0.000, E1  +307.505, E3 -101823.982}
SPL {X  -152.244, Y  +333.323, Z    +0.000, E1  +320.871, E3 -101840.793}
SPL {X  -158.218, Y  +358.753, Z    +0.000, E1  +336.397, E3 -101844.966}
SPL {X  -159.681, Y  +372.564, Z    +0.000, E1  +347.981, E3 -101846.017}
SPL {X  -159.987, Y  +381.561, Z    +0.000, E1  +356.806, E3 -101846.314}
SPL {X  -159.990, Y  +384.668, Z    +0.000, E1  +360.183, E3 -101846.339}
SPL {X  -159.990, Y  +387.837, Z    +0.000, E1  +367.342, E3 -101846.380}
SPL {X  -159.990, Y  +393.084, Z    +0.000, E1  +380.137, E3 -101846.590}
SPL {X  -159.990, Y  +401.914, Z    +0.000, E1  +400.147, E3 -101847.283}
SPL {X  -159.990, Y  +414.609, Z    +0.000, E1  +416.791, E3 -101849.020}
SPL {X  -159.990, Y  +464.476, Z    +0.000, E1  +431.765, E3 -101861.821}
SPL {X  -157.643, Y  +698.802, Z    +0.000, E1  +434.751, E3 -101964.836}
SPL {X  -154.470, Y  +713.164, Z    +0.000, E1  +434.425, E3 -101976.425}
SPL {X  -152.098, Y  +721.129, Z    +0.000, E1  +434.190, E3 -101983.397}
SPL {X  -148.128, Y  +731.956, Z    +0.000, E1  +433.814, E3 -101993.478}
SPL {X  -143.804, Y  +741.622, Z    +0.000, E1  +433.324, E3 -102003.254}
SPL {X  -140.603, Y  +747.839, Z    +0.000, E1  +432.964, E3 -102009.769}
SPL {X  -137.184, Y  +753.824, Z    +0.000, E1  +432.574, E3 -102016.206}
SPL {X  -133.762, Y  +759.276, Z    +0.000, E1  +432.150, E3 -102022.260}
SPL {X  -130.927, Y  +763.451, Z    +0.000, E1  +431.785, E3 -102026.954}
SPL {X  -128.105, Y  +767.343, Z    +0.000, E1  +431.419, E3 -102031.343}
SPL {X  -124.554, Y  +771.914, Z    +0.000, E1  +430.935, E3 -102036.514}
SPL {X  -120.892, Y  +776.295, Z    +0.000, E1  +430.404, E3 -102041.398}
SPL {X  -118.039, Y  +779.498, Z    +0.000, E1  +429.949, E3 -102044.916}
SPL {X   -71.924, Y  +814.412, Z    +0.000, E1  +415.124, E3 -102199.672}
ENDSPLINE

SPLINE
SPL {X  -132.255, Y  +761.530, Z    +0.000, E1  +413.203, E3 -102362.842}
SPL {X  -150.415, Y  +726.018, Z    +0.000, E1  +402.769, E3 -102376.346}
SPL {X  -156.153, Y  +706.328, Z    +0.000, E1  +392.414, E3 -102380.038}
SPL {X  -159.178, Y  +687.603, Z    +0.000, E1  +378.267, E3 -102382.016}
SPL {X  -159.974, Y  +673.783, Z    +0.000, E1  +364.843, E3 -102382.637}
SPL {X  -159.990, Y  +669.500, Z    +0.000, E1  +360.000, E3 -102382.685}
SPL {X  -159.990, Y  +667.470, Z    +0.000, E1  +355.588, E3 -102382.703}
SPL {X  -159.990, Y  +662.995, Z    +0.000, E1  +343.976, E3 -102382.819}
SPL {X  -159.990, Y  +658.179, Z    +0.000, E1  +331.312, E3 -102383.056}
SPL {X  -159.990, Y  +652.822, Z    +0.000, E1  +319.345, E3 -102383.471}
SPL {X  -159.990, Y  +646.185, Z    +0.000, E1  +308.728, E3 -102384.210}
SPL {X  -159.990, Y  +636.375, Z    +0.000, E1  +299.286, E3 -102385.649}
SPL {X  -159.990, Y  +617.374, Z    +0.000, E1  +291.478, E3 -102389.975}
SPL {X  -159.990, Y  +579.000, Z    +0.000, E1  +286.931, E3 -102401.434}
SPL {X  -157.725, Y  +355.675, Z    +0.000, E1  +284.959, E3 -102498.393}
SPL {X  -142.593, Y  +309.947, Z    +0.000, E1  +282.426, E3 -102492.056}
SPL {X  -142.198, Y  +309.176, Z    +0.000, E1  +283.218, E3 -102500.865}
ENDSPLINE

SPLINE
SPL {X  -142.352, Y  +309.474, Z    +0.000, E1  +284.206, E3 -102510.558}
ENDSPLINE

SPLINE
SPL {X  -141.553, Y  +307.937, Z    +0.000, E1  +285.290, E3 -102521.574}
SPL {X  -140.562, Y  +306.086, Z    +0.000, E1  +286.440, E3 -102532.268}
SPL {X  -138.743, Y  +302.832, Z    +0.000, E1  +287.062, E3 -102539.065}
SPL {X  -135.531, Y  +297.482, Z    +0.000, E1  +287.444, E3 -102544.900}
SPL {X  -132.271, Y  +292.493, Z    +0.000, E1  +287.844, E3 -102550.418}
SPL {X  -128.837, Y  +287.643, Z    +0.000, E1  +288.283, E3 -102555.856}
SPL {X  -125.941, Y  +283.830, Z    +0.000, E1  +288.683, E3 -102560.156}
SPL {X  -124.080, Y  +281.501, Z    +0.000, E1  +288.943, E3 -102562.766}
SPL {X  -120.791, Y  +277.589, Z    +0.000, E1  +289.397, E3 -102567.091}
SPL {X   -74.058, Y  +240.683, Z    +0.000, E1  +305.011, E3 -102724.154}
ENDSPLINE

SPLINE
SPL {X  -130.401, Y  +289.805, Z    +0.000, E1  +307.505, E3 -102881.125}
SPL {X  -148.502, Y  +322.968, Z    +0.000, E1  +316.497, E3 -102895.445}
SPL {X  -154.800, Y  +342.080, Z    +0.000, E1  +325.471, E3 -102899.749}
SPL {X  -158.218, Y  +358.753, Z    +0.000, E1  +336.397, E3 -102902.108}
SPL {X  -159.681, Y  +372.564, Z    +0.000, E1  +347.981, E3 -102903.160}
SPL {X  -159.987, Y  +381.561, Z    +0.000, E1  +356.806, E3 -102903.456}
SPL {X  -159.990, Y  +384.668, Z    +0.000, E1  +360.183, E3 -102903.482}
SPL {X  -159.990, Y  +387.837, Z    +0.000, E1  +367.342, E3 -102903.523}
SPL {X  -159.990, Y  +393.084, Z    +0.000, E1  +380.137, E3 -102903.733}
SPL {X  -159.990, Y  +401.914, Z    +0.000, E1  +400.147, E3 -102904.426}
SPL {X  -159.990, Y  +414.609, Z    +0.000, E1  +416.791, E3 -102906.163}
SPL {X  -159.990, Y  +464.476, Z    +0.000, E1  +431.765, E3 -102918.964}
SPL {X  -157.643, Y  +698.802, Z    +0.000, E1  +434.751, E3 -103021.979}
SPL {X  -154.470, Y  +713.164, Z    +0.000, E1  +434.425, E3 -103033.568}
SPL {X  -151.032, Y  +724.285, Z    +0.000, E1  +434.102, E3 -103043.371}
SPL {X  -147.134, Y  +734.337, Z    +0.000, E1  +433.686, E3 -103053.009}
SPL {X  -143.804, Y  +741.622, Z    +0.000, E1  +433.324, E3 -103060.397}
SPL {X  -140.603, Y  +747.839, Z    +0.000, E1  +432.964, E3 -103066.912}
SPL {X  -137.184, Y  +753.824, Z    +0.000, E1  +432.574, E3 -103073.349}
SPL {X  -133.762, Y  +759.276, Z    +0.000, E1  +432.150, E3 -103079.403}
SPL {X  -130.927, Y  +763.451, Z    +0.000, E1  +431.785, E3 -103084.097}
SPL {X  -128.105, Y  +767.343, Z    +0.000, E1  +431.419, E3 -103088.486}
SPL {X  -124.554, Y  +771.914, Z    +0.000, E1  +430.935, E3 -103093.657}
SPL {X  -120.892, Y  +776.295, Z    +0.000, E1  +430.404, E3 -103098.541}
SPL {X  -118.039, Y  +779.498, Z    +0.000, E1  +429.949, E3 -103102.059}
SPL {X   -71.924, Y  +814.412, Z    +0.000, E1  +415.124, E3 -103256.815}
ENDSPLINE

SPLINE
SPL {X  -132.255, Y  +761.530, Z    +0.000, E1  +413.203, E3 -103419.984}
SPL {X  -150.415, Y  +726.018, Z    +0.000, E1  +402.769, E3 -103433.488}
SPL {X  -156.153, Y  +706.328, Z    +0.000, E1  +392.414, E3 -103437.181}
SPL {X  -159.178, Y  +687.603, Z    +0.000, E1  +378.267, E3 -103439.158}
SPL {X  -159.974, Y  +673.783, Z    +0.000, E1  +364.843, E3 -103439.780}
SPL {X  -159.990, Y  +669.500, Z    +0.000, E1  +360.000, E3 -103439.828}
SPL {X  -159.990, Y  +667.470, Z    +0.000, E1  +355.588, E3 -103439.846}
SPL {X  -159.990, Y  +662.995, Z    +0.000, E1  +343.976, E3 -103439.962}
SPL {X  -159.990, Y  +658.179, Z    +0.000, E1  +331.312, E3 -103440.199}
SPL {X  -159.990, Y  +652.822, Z    +0.000, E1  +319.345, E3 -103440.614}
SPL {X  -159.990, Y  +646.185, Z    +0.000, E1  +308.728, E3 -103441.352}
SPL {X  -159.990, Y  +636.375, Z    +0.000, E1  +299.286, E3 -103442.792}
SPL {X  -159.990, Y  +617.374, Z    +0.000, E1  +291.478, E3 -103447.118}
SPL {X  -159.990, Y  +579.000, Z    +0.000, E1  +286.931, E3 -103458.577}
SPL {X  -157.725, Y  +355.675, Z    +0.000, E1  +284.959, E3 -103555.536}
SPL {X  -142.593, Y  +309.947, Z    +0.000, E1  +282.426, E3 -103549.199}
SPL {X  -142.198, Y  +309.176, Z    +0.000, E1  +283.218, E3 -103558.008}
ENDSPLINE

SPLINE
SPL {X  -142.352, Y  +309.474, Z    +0.000, E1  +284.206, E3 -103567.701}
ENDSPLINE

SPLINE
SPL {X  -141.553, Y  +307.937, Z    +0.000, E1  +285.290, E3 -103578.717}
SPL {X  -140.562, Y  +306.086, Z    +0.000, E1  +286.440, E3 -103589.411}
SPL {X  -138.743, Y  +302.832, Z    +0.000, E1  +287.062, E3 -103596.208}
SPL {X  -135.531, Y  +297.482, Z    +0.000, E1  +287.444, E3 -103602.043}
SPL {X  -132.271, Y  +292.493, Z    +0.000, E1  +287.844, E3 -103607.561}
SPL {X  -128.837, Y  +287.643, Z    +0.000, E1  +288.283, E3 -103612.999}
SPL {X  -124.965, Y  +282.598, Z    +0.000, E1  +288.800, E3 -103618.661}
SPL {X  -120.791, Y  +277.589, Z    +0.000, E1  +289.397, E3 -103624.234}
SPL {X   -74.058, Y  +240.683, Z    +0.000, E1  +305.011, E3 -103781.297}
ENDSPLINE

SPLINE
SPL {X  -130.401, Y  +289.805, Z    +0.000, E1  +307.505, E3 -103938.267}
SPL {X  -148.502, Y  +322.968, Z    +0.000, E1  +316.497, E3 -103952.588}
SPL {X  -154.800, Y  +342.080, Z    +0.000, E1  +325.471, E3 -103956.891}
SPL {X  -158.218, Y  +358.753, Z    +0.000, E1  +336.397, E3 -103959.251}
SPL {X  -159.681, Y  +372.564, Z    +0.000, E1  +347.981, E3 -103960.303}
SPL {X  -159.987, Y  +381.561, Z    +0.000, E1  +356.806, E3 -103960.599}
SPL {X  -159.990, Y  +384.668, Z    +0.000, E1  +360.183, E3 -103960.625}
SPL {X  -159.990, Y  +387.837, Z    +0.000, E1  +367.342, E3 -103960.666}
SPL {X  -159.990, Y  +393.084, Z    +0.000, E1  +380.137, E3 -103960.876}
SPL {X  -159.990, Y  +401.914, Z    +0.000, E1  +400.147, E3 -103961.569}
SPL {X  -159.990, Y  +414.609, Z    +0.000, E1  +416.791, E3 -103963.306}
SPL {X  -159.990, Y  +464.476, Z    +0.000, E1  +431.765, E3 -103976.107}
SPL {X  -157.643, Y  +698.802, Z    +0.000, E1  +434.751, E3 -104079.122}
SPL {X  -154.470, Y  +713.164, Z    +0.000, E1  +434.425, E3 -104090.710}
SPL {X  -151.032, Y  +724.285, Z    +0.000, E1  +434.102, E3 -104100.514}
SPL {X  -147.134, Y  +734.337, Z    +0.000, E1  +433.686, E3 -104110.152}
SPL {X  -143.804, Y  +741.622, Z    +0.000, E1  +433.324, E3 -104117.540}
SPL {X  -140.603, Y  +747.839, Z    +0.000, E1  +432.964, E3 -104124.055}
SPL {X  -137.184, Y  +753.824, Z    +0.000, E1  +432.574, E3 -104130.492}
SPL {X  -133.762, Y  +759.276, Z    +0.000, E1  +432.150, E3 -104136.546}
SPL {X  -130.927, Y  +763.451, Z    +0.000, E1  +431.785, E3 -104141.240}
SPL {X  -128.105, Y  +767.343, Z    +0.000, E1  +431.419, E3 -104145.629}
SPL {X  -124.554, Y  +771.914, Z    +0.000, E1  +430.935, E3 -104150.800}
SPL {X  -120.892, Y  +776.295, Z    +0.000, E1  +430.404, E3 -104155.684}
SPL {X  -118.039, Y  +779.498, Z    +0.000, E1  +429.949, E3 -104159.202}
SPL {X   -71.966, Y  +814.391, Z    +0.000, E1  +415.783, E3 -104297.854}
ENDSPLINE

SPLINE
SPL {X  -117.449, Y  +780.140, Z    +0.000, E1  +415.491, E3 -104462.268}
SPL {X  -137.837, Y  +752.727, Z    +0.000, E1  +411.385, E3 -104481.756}
SPL {X  -150.415, Y  +726.018, Z    +0.000, E1  +402.769, E3 -104490.631}
SPL {X  -156.153, Y  +706.328, Z    +0.000, E1  +392.414, E3 -104494.323}
SPL {X  -159.178, Y  +687.603, Z    +0.000, E1  +378.267, E3 -104496.301}
SPL {X  -159.915, Y  +676.399, Z    +0.000, E1  +367.484, E3 -104496.871}
SPL {X  -159.990, Y  +669.381, Z    +0.000, E1  +359.965, E3 -104496.971}
SPL {X  -159.990, Y  +666.412, Z    +0.000, E1  +352.765, E3 -104497.003}
SPL {X  -159.990, Y  +662.995, Z    +0.000, E1  +343.976, E3 -104497.105}
SPL {X  -159.990, Y  +658.179, Z    +0.000, E1  +331.312, E3 -104497.342}
SPL {X  -159.990, Y  +652.822, Z    +0.000, E1  +319.345, E3 -104497.757}
SPL {X  -159.990, Y  +646.185, Z    +0.000, E1  +308.728, E3 -104498.495}
SPL {X  -159.990, Y  +632.371, Z    +0.000, E1  +297.040, E3 -104500.848}
SPL {X  -159.990, Y  +579.000, Z    +0.000, E1  +286.931, E3 -104515.720}
SPL {X  -157.725, Y  +355.675, Z    +0.000, E1  +284.959, E3 -104612.678}
SPL {X  -142.593, Y  +309.947, Z    +0.000, E1  +282.426, E3 -104606.342}
SPL {X  -142.198, Y  +309.176, Z    +0.000, E1  +283.218, E3 -104615.150}
ENDSPLINE

SPLINE
SPL {X  -142.352, Y  +309.474, Z    +0.000, E1  +284.206, E3 -104624.844}
ENDSPLINE

SPLINE
SPL {X  -141.553, Y  +307.937, Z    +0.000, E1  +285.290, E3 -104635.860}
SPL {X  -140.562, Y  +306.086, Z    +0.000, E1  +286.440, E3 -104646.554}
SPL {X  -138.743, Y  +302.832, Z    +0.000, E1  +287.062, E3 -104653.351}
SPL {X  -135.531, Y  +297.482, Z    +0.000, E1  +287.444, E3 -104659.186}
SPL {X  -132.271, Y  +292.493, Z    +0.000, E1  +287.844, E3 -104664.704}
SPL {X  -128.837, Y  +287.643, Z    +0.000, E1  +288.283, E3 -104670.142}
SPL {X  -125.941, Y  +283.830, Z    +0.000, E1  +288.683, E3 -104674.442}
SPL {X  -122.669, Y  +279.791, Z    +0.000, E1  +289.119, E3 -104678.935}
SPL {X  -119.730, Y  +276.380, Z    +0.000, E1  +289.584, E3 -104682.723}
SPL {X   -74.058, Y  +240.683, Z    +0.000, E1  +305.011, E3 -104838.439}
ENDSPLINE

SPLINE
SPL {X  -130.401, Y  +289.805, Z    +0.000, E1  +307.505, E3 -104995.410}
SPL {X  -148.502, Y  +322.968, Z    +0.000, E1  +316.497, E3 -105009.731}
SPL {X  -154.800, Y  +342.080, Z    +0.000, E1  +325.471, E3 -105014.034}
SPL {X  -158.218, Y  +358.753, Z    +0.000, E1  +336.397, E3 -105016.394}
SPL {X  -159.681, Y  +372.564, Z    +0.000, E1  +347.981, E3 -105017.446}
SPL {X  -159.987, Y  +381.561, Z    +0.000, E1  +356.806, E3 -105017.742}
SPL {X  -159.990, Y  +384.668, Z    +0.000, E1  +360.183, E3 -105017.768}
SPL {X  -159.990, Y  +387.837, Z    +0.000, E1  +367.342, E3 -105017.809}
SPL {X  -159.990, Y  +393.084, Z    +0.000, E1  +380.137, E3 -105018.018}
SPL {X  -159.990, Y  +401.914, Z    +0.000, E1  +400.147, E3 -105018.712}
SPL {X  -159.990, Y  +414.609, Z    +0.000, E1  +416.791, E3 -105020.449}
SPL {X  -159.990, Y  +464.476, Z    +0.000, E1  +431.765, E3 -105033.250}
SPL {X  -157.643, Y  +698.802, Z    +0.000, E1  +434.751, E3 -105136.265}
SPL {X  -154.470, Y  +713.164, Z    +0.000, E1  +434.425, E3 -105147.853}
SPL {X  -151.032, Y  +724.285, Z    +0.000, E1  +434.102, E3 -105157.657}
SPL {X  -147.134, Y  +734.337, Z    +0.000, E1  +433.686, E3 -105167.295}
SPL {X  -143.804, Y  +741.622, Z    +0.000, E1  +433.324, E3 -105174.682}
SPL {X  -140.603, Y  +747.839, Z    +0.000, E1  +432.964, E3 -105181.198}
SPL {X  -137.184, Y  +753.824, Z    +0.000, E1  +432.574, E3 -105187.635}
SPL {X  -133.762, Y  +759.276, Z    +0.000, E1  +432.150, E3 -105193.688}
SPL {X  -130.927, Y  +763.451, Z    +0.000, E1  +431.785, E3 -105198.383}
SPL {X  -128.105, Y  +767.343, Z    +0.000, E1  +431.419, E3 -105202.772}
SPL {X  -124.554, Y  +771.914, Z    +0.000, E1  +430.935, E3 -105207.943}
SPL {X  -120.892, Y  +776.295, Z    +0.000, E1  +430.404, E3 -105212.827}
SPL {X  -118.039, Y  +779.498, Z    +0.000, E1  +429.949, E3 -105216.345}
SPL {X   -71.924, Y  +814.412, Z    +0.000, E1  +415.124, E3 -105371.100}
ENDSPLINE

SPLINE
SPL {X  -132.255, Y  +761.530, Z    +0.000, E1  +413.203, E3 -105534.270}
SPL {X  -150.415, Y  +726.018, Z    +0.000, E1  +402.769, E3 -105547.774}
SPL {X  -156.153, Y  +706.328, Z    +0.000, E1  +392.414, E3 -105551.466}
SPL {X  -159.178, Y  +687.603, Z    +0.000, E1  +378.267, E3 -105553.444}
SPL {X  -159.974, Y  +673.783, Z    +0.000, E1  +364.843, E3 -105554.066}
SPL {X  -159.990, Y  +669.500, Z    +0.000, E1  +360.000, E3 -105554.114}
SPL {X  -159.990, Y  +667.470, Z    +0.000, E1  +355.588, E3 -105554.132}
SPL {X  -159.990, Y  +662.995, Z    +0.000, E1  +343.976, E3 -105554.248}
SPL {X  -159.990, Y  +658.179, Z    +0.000, E1  +331.312, E3 -105554.485}
SPL {X  -159.990, Y  +652.822, Z    +0.000, E1  +319.345, E3 -105554.899}
SPL {X  -159.990, Y  +646.185, Z    +0.000, E1  +308.728, E3 -105555.638}
SPL {X  -159.990, Y  +636.375, Z    +0.000, E1  +299.286, E3 -105557.078}
SPL {X  -159.990, Y  +617.374, Z    +0.000, E1  +291.478, E3 -105561.404}
SPL {X  -159.990, Y  +579.000, Z    +0.000, E1  +286.931, E3 -105572.863}
SPL {X  -157.725, Y  +355.675, Z    +0.000, E1  +284.959, E3 -105669.821}
SPL {X  -142.593, Y  +309.947, Z    +0.000, E1  +282.426, E3 -105663.485}
SPL {X  -142.198, Y  +309.176, Z    +0.000, E1  +283.218, E3 -105672.293}
ENDSPLINE

SPLINE
SPL {X  -142.352, Y  +309.474, Z    +0.000, E1  +284.206, E3 -105681.987}
ENDSPLINE

SPLINE
SPL {X  -141.553, Y  +307.937, Z    +0.000, E1  +285.290, E3 -105693.003}
SPL {X  -140.511, Y  +305.992, Z    +0.000, E1  +286.445, E3 -105703.797}
ENDSPLINE

SPLINE
SPL {X  -147.030, Y  +319.421, Z    +0.000, E1  +289.755, E3 -105722.112}
ENDSPLINE

SPLINE
SPL {X  -143.573, Y  +311.906, Z    +0.000, E1  +290.194, E3 -105730.687}
SPL {X  -139.693, Y  +304.508, Z    +0.000, E1  +290.699, E3 -105739.415}
SPL {X  -135.622, Y  +297.627, Z    +0.000, E1  +291.269, E3 -105747.823}
SPL {X  -131.165, Y  +290.889, Z    +0.000, E1  +291.906, E3 -105756.209}
SPL {X  -126.457, Y  +284.492, Z    +0.000, E1  +292.648, E3 -105764.294}
SPL {X  -123.432, Y  +280.710, Z    +0.000, E1  +293.170, E3 -105769.080}
SPL {X   -85.607, Y  +247.340, Z    +0.000, E1  +306.083, E3 -105910.801}
ENDSPLINE

SPLINE
SPL {X  -134.737, Y  +296.229, Z    +0.000, E1  +312.110, E3 -106053.574}
SPL {X  -154.917, Y  +342.531, Z    +0.000, E1  +328.797, E3 -106072.142}
SPL {X  -159.440, Y  +369.246, Z    +0.000, E1  +346.542, E3 -106076.041}
SPL {X  -159.987, Y  +381.470, Z    +0.000, E1  +357.024, E3 -106076.640}
SPL {X  -159.990, Y  +384.500, Z    +0.000, E1  +360.000, E3 -106076.673}
SPL {X  -159.990, Y  +386.323, Z    +0.000, E1  +363.079, E3 -106076.695}
SPL {X  -159.990, Y  +390.285, Z    +0.000, E1  +371.315, E3 -106076.816}
SPL {X  -159.990, Y  +394.559, Z    +0.000, E1  +380.770, E3 -106077.078}
SPL {X  -159.990, Y  +402.118, Z    +0.000, E1  +395.793, E3 -106077.869}
SPL {X  -159.990, Y  +415.193, Z    +0.000, E1  +412.724, E3 -106080.122}
SPL {X  -159.990, Y  +465.395, Z    +0.000, E1  +428.959, E3 -106095.210}
SPL {X  -159.990, Y  +657.157, Z    +0.000, E1  +432.499, E3 -106191.607}
SPL {X  -159.693, Y  +681.249, Z    +0.000, E1  +432.488, E3 -106208.001}
SPL {X  -157.599, Y  +699.059, Z    +0.000, E1  +432.249, E3 -106222.161}
SPL {X  -155.217, Y  +710.289, Z    +0.000, E1  +431.989, E3 -106232.177}
SPL {X  -152.611, Y  +719.527, Z    +0.000, E1  +431.702, E3 -106240.999}
SPL {X  -149.536, Y  +728.383, Z    +0.000, E1  +431.359, E3 -106249.978}
SPL {X  -146.250, Y  +736.367, Z    +0.000, E1  +430.965, E3 -106258.532}
SPL {X  -143.481, Y  +742.281, Z    +0.000, E1  +430.623, E3 -106265.128}
SPL {X  -140.071, Y  +748.811, Z    +0.000, E1  +430.193, E3 -106272.639}
SPL {X  -136.578, Y  +754.826, Z    +0.000, E1  +429.723, E3 -106279.769}
SPL {X  -133.265, Y  +760.028, Z    +0.000, E1  +429.258, E3 -106286.070}
SPL {X  -129.890, Y  +764.909, Z    +0.000, E1  +428.775, E3 -106292.040}
SPL {X  -125.802, Y  +770.346, Z    +0.000, E1  +428.156, E3 -106298.739}
SPL {X  -122.624, Y  +774.263, Z    +0.000, E1  +427.622, E3 -106303.562}
SPL {X   -84.435, Y  +807.395, Z    +0.000, E1  +415.948, E3 -106414.566}
ENDSPLINE

SPLINE
SPL {X  -119.703, Y  +777.650, Z    +0.000, E1  +411.831, E3 -106578.573}
SPL {X  -145.184, Y  +738.720, Z    +0.000, E1  +403.488, E3 -106605.131}
SPL {X  -156.175, Y  +706.232, Z    +0.000, E1  +388.819, E3 -106614.016}
SPL {X  -159.337, Y  +685.942, Z    +0.000, E1  +374.672, E3 -106616.567}
SPL {X  -159.962, Y  +674.468, Z    +0.000, E1  +364.846, E3 -106617.186}
SPL {X  -159.990, Y  +669.479, Z    +0.000, E1  +359.996, E3 -106617.260}
SPL {X  -159.990, Y  +667.035, Z    +0.000, E1  +355.461, E3 -106617.291}
SPL {X  -159.990, Y  +662.914, Z    +0.000, E1  +346.506, E3 -106617.430}
SPL {X  -159.990, Y  +658.254, Z    +0.000, E1  +335.847, E3 -106617.707}
SPL {X  -159.990, Y  +652.944, Z    +0.000, E1  +324.878, E3 -106618.211}
SPL {X  -159.990, Y  +642.509, Z    +0.000, E1  +309.910, E3 -106619.783}
SPL {X  -159.990, Y  +618.566, Z    +0.000, E1  +295.881, E3 -106625.953}
SPL {X  -159.990, Y  +582.261, Z    +0.000, E1  +290.657, E3 -106639.439}
SPL {X  -159.990, Y  +414.423, Z    +0.000, E1  +288.398, E3 -106730.222}
SPL {X  -159.990, Y  +400.357, Z    +0.000, E1  +288.396, E3 -106740.133}
SPL {X  -159.990, Y  +385.723, Z    +0.000, E1  +288.390, E3 -106750.424}
SPL {X  -159.404, Y  +368.814, Z    +0.000, E1  +288.444, E3 -106762.953}
SPL {X  -157.440, Y  +354.048, Z    +0.000, E1  +288.658, E3 -106775.426}
SPL {X  -155.538, Y  +345.018, Z    +0.000, E1  +288.891, E3 -106783.819}
SPL {X  -155.351, Y  +344.251, Z    +0.000, E1  +289.996, E3 -106794.536}
SPL {X  -150.579, Y  +328.438, Z    +0.000, E1  +289.626, E3 -106802.921}
SPL {X  -146.933, Y  +319.195, Z    +0.000, E1  +289.770, E3 -106810.612}
SPL {X  -143.573, Y  +311.906, Z    +0.000, E1  +290.194, E3 -106818.922}
SPL {X  -139.693, Y  +304.508, Z    +0.000, E1  +290.699, E3 -106827.650}
SPL {X  -135.622, Y  +297.627, Z    +0.000, E1  +291.269, E3 -106836.059}
SPL {X  -132.531, Y  +292.877, Z    +0.000, E1  +291.734, E3 -106841.994}
SPL {X  -128.822, Y  +287.623, Z    +0.000, E1  +292.271, E3 -106848.568}
SPL {X  -124.502, Y  +282.021, Z    +0.000, E1  +292.965, E3 -106855.642}
SPL {X   -85.607, Y  +247.340, Z    +0.000, E1  +306.083, E3 -106999.036}
ENDSPLINE

SPLINE
SPL {X  -134.737, Y  +296.229, Z    +0.000, E1  +312.110, E3 -107141.809}
SPL {X  -154.917, Y  +342.531, Z    +0.000, E1  +328.797, E3 -107160.377}
SPL {X  -159.440, Y  +369.246, Z    +0.000, E1  +346.542, E3 -107164.276}
SPL {X  -159.987, Y  +381.470, Z    +0.000, E1  +357.024, E3 -107164.875}
SPL {X  -159.990, Y  +384.500, Z    +0.000, E1  +360.000, E3 -107164.908}
SPL {X  -159.990, Y  +386.323, Z    +0.000, E1  +363.079, E3 -107164.930}
SPL {X  -159.990, Y  +390.285, Z    +0.000, E1  +371.315, E3 -107165.051}
SPL {X  -159.990, Y  +394.559, Z    +0.000, E1  +380.770, E3 -107165.313}
SPL {X  -159.990, Y  +402.118, Z    +0.000, E1  +395.793, E3 -107166.105}
SPL {X  -159.990, Y  +415.193, Z    +0.000, E1  +412.724, E3 -107168.357}
SPL {X  -159.990, Y  +465.395, Z    +0.000, E1  +428.959, E3 -107183.446}
SPL {X  -159.990, Y  +652.170, Z    +0.000, E1  +432.485, E3 -107276.541}
SPL {X  -159.990, Y  +670.864, Z    +0.000, E1  +432.509, E3 -107288.989}
SPL {X  -159.251, Y  +686.856, Z    +0.000, E1  +432.412, E3 -107300.531}
SPL {X  -157.599, Y  +699.059, Z    +0.000, E1  +432.249, E3 -107310.396}
SPL {X  -155.217, Y  +710.289, Z    +0.000, E1  +431.989, E3 -107320.413}
SPL {X  -152.611, Y  +719.527, Z    +0.000, E1  +431.702, E3 -107329.234}
SPL {X  -149.536, Y  +728.383, Z    +0.000, E1  +431.359, E3 -107338.213}
SPL {X  -146.250, Y  +736.367, Z    +0.000, E1  +430.965, E3 -107346.767}
SPL {X  -143.481, Y  +742.281, Z    +0.000, E1  +430.623, E3 -107353.363}
SPL {X  -140.071, Y  +748.811, Z    +0.000, E1  +430.193, E3 -107360.875}
SPL {X  -136.578, Y  +754.826, Z    +0.000, E1  +429.723, E3 -107368.004}
SPL {X  -132.176, Y  +761.646, Z    +0.000, E1  +429.128, E3 -107376.247}
SPL {X  -127.941, Y  +767.561, Z    +0.000, E1  +428.475, E3 -107383.555}
SPL {X  -123.778, Y  +772.869, Z    +0.000, E1  +427.843, E3 -107390.063}
SPL {X   -84.435, Y  +807.395, Z    +0.000, E1  +415.948, E3 -107502.802}
ENDSPLINE

SPLINE
SPL {X  -119.703, Y  +777.650, Z    +0.000, E1  +411.831, E3 -107666.808}
SPL {X  -145.184, Y  +738.720, Z    +0.000, E1  +403.488, E3 -107693.366}
SPL {X  -156.175, Y  +706.232, Z    +0.000, E1  +388.819, E3 -107702.251}
SPL {X  -159.337, Y  +685.942, Z    +0.000, E1  +374.672, E3 -107704.802}
SPL {X  -159.962, Y  +674.468, Z    +0.000, E1  +364.846, E3 -107705.421}
SPL {X  -159.990, Y  +669.479, Z    +0.000, E1  +359.996, E3 -107705.495}
SPL {X  -159.990, Y  +667.035, Z    +0.000, E1  +355.461, E3 -107705.526}
SPL {X  -159.990, Y  +662.914, Z    +0.000, E1  +346.506, E3 -107705.665}
SPL {X  -159.990, Y  +658.254, Z    +0.000, E1  +335.847, E3 -107705.943}
SPL {X  -159.990, Y  +650.381, Z    +0.000, E1  +320.607, E3 -107706.794}
SPL {X  -159.990, Y  +638.701, Z    +0.000, E1  +306.047, E3 -107708.680}
SPL {X  -159.990, Y  +618.566, Z    +0.000, E1  +295.881, E3 -107714.188}
SPL {X  -159.990, Y  +582.261, Z    +0.000, E1  +290.657, E3 -107727.674}
SPL {X  -159.990, Y  +414.423, Z    +0.000, E1  +288.398, E3 -107818.457}
SPL {X  -159.990, Y  +400.357, Z    +0.000, E1  +288.396, E3 -107828.368}
SPL {X  -159.990, Y  +385.723, Z    +0.000, E1  +288.390, E3 -107838.659}
SPL {X  -159.404, Y  +368.814, Z    +0.000, E1  +288.444, E3 -107851.188}
SPL {X  -157.440, Y  +354.048, Z    +0.000, E1  +288.658, E3 -107863.662}
SPL {X  -155.889, Y  +346.508, Z    +0.000, E1  +289.539, E3 -107877.210}
SPL {X  -154.332, Y  +340.328, Z    +0.000, E1  +289.976, E3 -107885.438}
SPL {X  -150.579, Y  +328.438, Z    +0.000, E1  +289.626, E3 -107891.156}
SPL {X  -146.933, Y  +319.195, Z    +0.000, E1  +289.770, E3 -107898.847}
SPL {X  -143.573, Y  +311.906, Z    +0.000, E1  +290.194, E3 -107907.158}
SPL {X  -139.693, Y  +304.508, Z    +0.000, E1  +290.699, E3 -107915.886}
SPL {X  -135.622, Y  +297.627, Z    +0.000, E1  +291.269, E3 -107924.294}
SPL {X  -131.165, Y  +290.889, Z    +0.000, E1  +291.906, E3 -107932.679}
SPL {X  -126.457, Y  +284.492, Z    +0.000, E1  +292.648, E3 -107940.765}
SPL {X  -123.432, Y  +280.710, Z    +0.000, E1  +293.170, E3 -107945.550}
SPL {X   -85.607, Y  +247.340, Z    +0.000, E1  +306.083, E3 -108087.272}
ENDSPLINE

SPLINE
SPL {X  -134.737, Y  +296.229, Z    +0.000, E1  +312.110, E3 -108230.045}
SPL {X  -153.211, Y  +336.421, Z    +0.000, E1  +325.738, E3 -108247.252}
SPL {X  -158.240, Y  +358.900, Z    +0.000, E1  +338.911, E3 -108251.458}
SPL {X  -159.854, Y  +375.896, Z    +0.000, E1  +352.019, E3 -108252.924}
SPL {X  -159.990, Y  +384.670, Z    +0.000, E1  +360.079, E3 -108253.145}
SPL {X  -159.990, Y  +389.248, Z    +0.000, E1  +368.879, E3 -108253.249}
SPL {X  -159.990, Y  +394.559, Z    +0.000, E1  +380.770, E3 -108253.548}
SPL {X  -159.990, Y  +402.118, Z    +0.000, E1  +395.793, E3 -108254.340}
SPL {X  -159.990, Y  +415.193, Z    +0.000, E1  +412.724, E3 -108256.592}
SPL {X  -159.990, Y  +465.395, Z    +0.000, E1  +428.959, E3 -108271.681}
SPL {X  -159.990, Y  +657.157, Z    +0.000, E1  +432.499, E3 -108368.078}
SPL {X  -159.693, Y  +681.249, Z    +0.000, E1  +432.488, E3 -108384.472}
SPL {X  -157.599, Y  +699.059, Z    +0.000, E1  +432.249, E3 -108398.631}
SPL {X  -155.217, Y  +710.289, Z    +0.000, E1  +431.989, E3 -108408.648}
SPL {X  -152.611, Y  +719.527, Z    +0.000, E1  +431.702, E3 -108417.469}
SPL {X  -149.536, Y  +728.383, Z    +0.000, E1  +431.359, E3 -108426.449}
SPL {X  -146.250, Y  +736.367, Z    +0.000, E1  +430.965, E3 -108435.003}
SPL {X  -143.481, Y  +742.281, Z    +0.000, E1  +430.623, E3 -108441.598}
SPL {X  -140.071, Y  +748.811, Z    +0.000, E1  +430.193, E3 -108449.110}
SPL {X  -136.578, Y  +754.826, Z    +0.000, E1  +429.723, E3 -108456.239}
SPL {X  -133.265, Y  +760.028, Z    +0.000, E1  +429.258, E3 -108462.540}
SPL {X  -129.890, Y  +764.909, Z    +0.000, E1  +428.775, E3 -108468.511}
SPL {X  -125.802, Y  +770.346, Z    +0.000, E1  +428.156, E3 -108475.210}
SPL {X  -122.624, Y  +774.263, Z    +0.000, E1  +427.622, E3 -108480.033}
SPL {X   -84.435, Y  +807.395, Z    +0.000, E1  +415.948, E3 -108591.037}
ENDSPLINE

SPLINE
SPL {X  -119.703, Y  +777.650, Z    +0.000, E1  +411.831, E3 -108755.044}
SPL {X  -145.184, Y  +738.720, Z    +0.000, E1  +403.488, E3 -108781.602}
SPL {X  -154.467, Y  +713.173, Z    +0.000, E1  +392.658, E3 -108789.197}
SPL {X  -157.530, Y  +699.446, Z    +0.000, E1  +384.482, E3 -108791.613}
SPL {X  -159.337, Y  +685.942, Z    +0.000, E1  +374.672, E3 -108793.038}
SPL {X  -159.962, Y  +674.468, Z    +0.000, E1  +364.846, E3 -108793.656}
SPL {X  -159.990, Y  +669.479, Z    +0.000, E1  +359.996, E3 -108793.731}
SPL {X  -159.990, Y  +667.035, Z    +0.000, E1  +355.461, E3 -108793.761}
SPL {X  -159.990, Y  +662.914, Z    +0.000, E1  +346.506, E3 -108793.900}
SPL {X  -159.990, Y  +658.254, Z    +0.000, E1  +335.847, E3 -108794.178}
SPL {X  -159.990, Y  +652.944, Z    +0.000, E1  +324.878, E3 -108794.681}
SPL {X  -159.990, Y  +642.509, Z    +0.000, E1  +309.910, E3 -108796.253}
SPL {X  -159.990, Y  +618.566, Z    +0.000, E1  +295.881, E3 -108802.424}
SPL {X  -159.990, Y  +582.261, Z    +0.000, E1  +290.657, E3 -108815.909}
SPL {X  -159.990, Y  +406.555, Z    +0.000, E1  +288.365, E3 -108912.156}
SPL {X  -159.990, Y  +385.723, Z    +0.000, E1  +288.390, E3 -108926.894}
SPL {X  -159.700, Y  +372.863, Z    +0.000, E1  +288.430, E3 -108936.300}
SPL {X  -158.535, Y  +360.970, Z    +0.000, E1  +288.540, E3 -108945.871}
SPL {X  -156.277, Y  +348.230, Z    +0.000, E1  +288.789, E3 -108957.214}
SPL {X  -155.351, Y  +344.251, Z    +0.000, E1  +289.996, E3 -108971.006}
SPL {X  -150.579, Y  +328.438, Z    +0.000, E1  +289.626, E3 -108979.392}
SPL {X  -146.933, Y  +319.195, Z    +0.000, E1  +289.770, E3 -108987.082}
SPL {X  -143.573, Y  +311.906, Z    +0.000, E1  +290.194, E3 -108995.393}
SPL {X  -140.547, Y  +306.057, Z    +0.000, E1  +290.601, E3 -109002.285}
SPL {X  -137.438, Y  +300.600, Z    +0.000, E1  +291.016, E3 -109008.879}
SPL {X  -133.397, Y  +294.172, Z    +0.000, E1  +291.584, E3 -109016.814}
SPL {X  -128.822, Y  +287.623, Z    +0.000, E1  +292.271, E3 -109025.039}
SPL {X  -124.502, Y  +282.021, Z    +0.000, E1  +292.965, E3 -109032.112}
SPL {X   -85.607, Y  +247.340, Z    +0.000, E1  +306.083, E3 -109175.507}
ENDSPLINE

SPLINE
SPL {X  -119.557, Y  +276.184, Z    +0.000, E1  +308.968, E3 -109299.044}
SPL {X  -138.294, Y  +302.054, Z    +0.000, E1  +313.424, E3 -109322.366}
SPL {X  -153.211, Y  +336.421, Z    +0.000, E1  +325.738, E3 -109335.488}
SPL {X  -158.240, Y  +358.900, Z    +0.000, E1  +338.911, E3 -109339.693}
SPL {X  -159.674, Y  +372.451, Z    +0.000, E1  +349.222, E3 -109340.989}
SPL {X  -159.987, Y  +381.470, Z    +0.000, E1  +357.024, E3 -109341.346}
SPL {X  -159.990, Y  +384.761, Z    +0.000, E1  +360.257, E3 -109341.381}
SPL {X  -159.990, Y  +389.248, Z    +0.000, E1  +368.879, E3 -109341.485}
SPL {X  -159.990, Y  +394.559, Z    +0.000, E1  +380.770, E3 -109341.784}
SPL {X  -159.990, Y  +402.118, Z    +0.000, E1  +395.793, E3 -109342.575}
SPL {X  -159.990, Y  +415.193, Z    +0.000, E1  +412.724, E3 -109344.828}
SPL {X  -159.990, Y  +465.395, Z    +0.000, E1  +428.959, E3 -109359.916}
SPL {X  -159.990, Y  +657.157, Z    +0.000, E1  +432.499, E3 -109456.313}
SPL {X  -159.947, Y  +675.227, Z    +0.000, E1  +432.487, E3 -109468.473}
SPL {X  -159.251, Y  +686.856, Z    +0.000, E1  +432.412, E3 -109477.001}
SPL {X  -157.599, Y  +699.059, Z    +0.000, E1  +432.249, E3 -109486.867}
SPL {X  -155.217, Y  +710.289, Z    +0.000, E1  +431.989, E3 -109496.883}
SPL {X  -152.611, Y  +719.527, Z    +0.000, E1  +431.702, E3 -109505.705}
SPL {X  -149.536, Y  +728.383, Z    +0.000, E1  +431.359, E3 -109514.684}
SPL {X  -146.250, Y  +736.367, Z    +0.000, E1  +430.965, E3 -109523.238}
SPL {X  -143.481, Y  +742.281, Z    +0.000, E1  +430.623, E3 -109529.833}
SPL {X  -140.071, Y  +748.811, Z    +0.000, E1  +430.193, E3 -109537.345}
SPL {X  -136.578, Y  +754.826, Z    +0.000, E1  +429.723, E3 -109544.475}
SPL {X  -133.265, Y  +760.028, Z    +0.000, E1  +429.258, E3 -109550.775}
SPL {X  -129.890, Y  +764.909, Z    +0.000, E1  +428.775, E3 -109556.746}
SPL {X  -125.802, Y  +770.346, Z    +0.000, E1  +428.156, E3 -109563.445}
SPL {X  -122.624, Y  +774.263, Z    +0.000, E1  +427.622, E3 -109568.268}
SPL {X   -84.435, Y  +807.395, Z    +0.000, E1  +415.948, E3 -109679.272}
ENDSPLINE

